	20:	
		sState := CONCAT(UDINT_TO_STRING(nState) ,' - Alaphelyzetfelvétel - Robot bekapcsolása');
		RobotOut.Control.bImmediateStop := TRUE;
		RobotOut.Control.bHold := TRUE;
		RobotOut.Control.bSafeSpeed := TRUE;
		RobotOut.Control.bEnable := TRUE;
		IF RobotIn.Status.bFault AND NOT RobotOut.Control.bReset THEN
			RobotOut.Control.bReset := TRUE;	// Ha hiba van -> Reset
		END_IF
		nState := nState + 20;

	40:
		sState := CONCAT(UDINT_TO_STRING(nState) ,' - Alaphelyzet felvétel - Robot hibatörlés');	
		IF tResetFault.Q THEN
			RobotOut.Control.bReset := FALSE;
		END_IF
		IF NOT RobotOut.Control.bReset AND NOT RobotIn.Status.bFault THEN
			nState := nState + 20;
		END_IF

	60:
		sState := CONCAT(UDINT_TO_STRING(nState) ,' - Alaphelyzet felvétel - Várakozás Robot hibatörlésre');	
		IF RobotIn.Status.bCommandEnable AND NOT RobotIn.Status.bFault THEN
			nState := nState + 20;
		END_IF
		
	80:
		sState := CONCAT(UDINT_TO_STRING(nState) ,' - Alaphelyzet felvétel - Robot Cycle Stop');
		RobotOut.Control.bCycleStop := TRUE;
		IF tStopCycle.Q THEN
			RobotOut.Control.bCycleStop := FALSE;
			nState := nState + 20;
		END_IF
	
	100:
		sState := CONCAT(UDINT_TO_STRING(nState) ,' - Alaphelyzet felvétel - Robot Cycle Start');
		RobotOut.Control.bStart := TRUE;
		IF tStartCycle.Q THEN
			RobotOut.Control.bStart := FALSE;
			nState := nState + 20;
		END_IF
		
	120: 
		sState := CONCAT(UDINT_TO_STRING(nState) ,' - Alaphelyzet felvétel - Várakozás Robot Cycle Start-ra');
		IF RobotIn.Status.bBusy AND RobotIn.Status.bProgramEnd THEN
			nState := nState + 20;
		END_IF
		
	140:
		sState := CONCAT(UDINT_TO_STRING(nState) ,' - Alaphelyzet felvétel - Alaphelyzet felvétel - Robot Busy');
		IF RobotIn.Status.bBusy THEN
			RobotOut.Control.bProdStart := TRUE;
			nState := nState + 20;
		END_IF
		
	160:
		sState := CONCAT(UDINT_TO_STRING(nState) ,' - Alaphelyzet felvétel - Robot alaphelyzetbe küldése');	
		RobotOut.Control.nProgramNumber := TO_BYTE(E_Kardex_Robot_Programs.Home);
		IF RobotOut.Control.nProgramNumber = RobotIn.Status.nProgramNumber THEN
			RobotOut.Control.nProgramNumber := 0;
			nState := nState + 20;
		END_IF
		
	180:
		sState := CONCAT(UDINT_TO_STRING(nState) ,' - Alaphelyzet felvétel - Várakozás a robotprogram végére.');	
		IF RobotIn.Status.bProgramEnd AND NOT RobotIn.Status.bProgramRun THEN
			nState := nState + 20;
		END_IF
		
	200:
		nState := 10000;
		 
(* Alaphelyzet *********************************************************************)
	10000:
		sState := CONCAT(UDINT_TO_STRING(nState) ,' - Alaphelyzet - Várakozás parancsra');
		IF eCommand = E_Kardex_Robot_Command.NoCommand THEN
			bReady := TRUE;
			bBusy := FALSE;
			bDone := FALSE;
		ELSE
			bReady := TRUE;
			bBusy := TRUE;
			bDone := FALSE;
			IF eCommand = E_Kardex_Robot_Command.Home THEN			
				nState := 11000;	
			ELSIF eCommand = E_Kardex_Robot_Command.Wait THEN	
				nState := 12000;
			ELSIF eCommand = E_Kardex_Robot_Command.Service THEN	
				nState := 13000;
			ELSIF eCommand = E_Kardex_Robot_Command.Measurement_Kardex THEN	
				nState := 14000;
			ELSIF eCommand = E_Kardex_Robot_Command.Pick_Up_Kardex THEN	
				nState := 15000;
			ELSIF eCommand = E_Kardex_Robot_Command.Put_Down_Kardex THEN	
				nState := 16000;
			ELSIF eCommand = E_Kardex_Robot_Command.Pick_Up_Mir THEN	
				nState := 17000;
			ELSIF eCommand = E_Kardex_Robot_Command.Put_Down_Mir THEN	
				nState := 18000;
			ELSIF eCommand = E_Kardex_Robot_Command.Pick_Up_Puffer THEN	
				nState := 19000;
			ELSIF eCommand = E_Kardex_Robot_Command.Put_Down_Puffer THEN	
				nState := 20000;
			ELSIF eCommand = E_Kardex_Robot_Command.Pick_Up_Strip THEN	
				nState := 21000;
			ELSIF eCommand = E_Kardex_Robot_Command.Put_Down_Strip THEN	
				nState := 22000;
			ELSIF eCommand = E_Kardex_Robot_Command.Rotate_In_Strip_3 THEN	
				nState := 23000;
			END_IF
		END_IF

{region "Move to Home"} 
	(*-----=== Move to home program végrehajtása ===-----*)
	11000:	
		sState := CONCAT(UDINT_TO_STRING(nState) ,' - Robot alaphelyzetbe küldése');	
		RobotOut.Control.nProgramNumber := TO_BYTE(E_Kardex_Robot_Programs.Home);
		IF RobotOut.Control.nProgramNumber = RobotIn.Status.nProgramNumber THEN
			RobotOut.Control.nProgramNumber := 0;
			nState := nState + 20;
		END_IF
		
	11020:
		sState := CONCAT(UDINT_TO_STRING(nState) ,' - Várakozás a robotprogram végére.');	
		IF RobotIn.Status.bProgramEnd AND NOT RobotIn.Status.bProgramRun THEN
			nState := nState + 20;
		END_IF
		
	11040:
		sState := CONCAT(UDINT_TO_STRING(nState) ,' - Várakozás mozgásparancs törlésére.');
		bReady := TRUE;
		bBusy := FALSE;
		bDone := TRUE;
		IF eCommand = E_Kardex_Robot_Command.NoCommand THEN
			nState := 10000;
		END_IF
{endregion}
	 
{region "Move to Wait"}
	(*-----=== Move to wait program végrehajtása ===-----*)
	12000:	
		sState := CONCAT(UDINT_TO_STRING(nState) ,' - Robot várakozó pozícióba küldése');	
		RobotOut.Control.nProgramNumber := TO_BYTE(E_Kardex_Robot_Programs.Park);
		IF RobotOut.Control.nProgramNumber = RobotIn.Status.nProgramNumber THEN
			RobotOut.Control.nProgramNumber := 0;
			nState := nState + 20;
		END_IF
		
	12020:
		sState := CONCAT(UDINT_TO_STRING(nState) ,' - Várakozás a robotprogram végére.');	
		IF RobotIn.Status.bProgramEnd AND NOT RobotIn.Status.bProgramRun THEN
			nState := nState + 20;
		END_IF
		
	12040:
		sState := CONCAT(UDINT_TO_STRING(nState) ,' - Várakozás mozgásparancs törlésére.');
		bReady := TRUE;
		bBusy := FALSE;
		bDone := TRUE;
		IF eCommand = E_Kardex_Robot_Command.NoCommand THEN
			nState := 10000;
		END_IF
{endregion}
	 
{region "Move to Service"}
	(*-----=== Move to service program végrehajtása ===-----*)
	13000:	
		sState := CONCAT(UDINT_TO_STRING(nState) ,' - Robot szervíz pozícióba küldése');	
		RobotOut.Control.nProgramNumber := TO_BYTE(E_Kardex_Robot_Programs.Service);
		IF RobotOut.Control.nProgramNumber = RobotIn.Status.nProgramNumber THEN
			RobotOut.Control.nProgramNumber := 0;
			nState := nState + 20;
		END_IF
		
	13020:
		sState := CONCAT(UDINT_TO_STRING(nState) ,' - Várakozás a robotprogram végére.');	
		IF RobotIn.Status.bProgramEnd AND NOT RobotIn.Status.bProgramRun THEN
			nState := nState + 20;
		END_IF
		
	13040:
		sState := CONCAT(UDINT_TO_STRING(nState) ,' - Várakozás mozgásparancs törlésére.');
		bReady := TRUE;
		bBusy := FALSE;
		bDone := TRUE;
		IF eCommand = E_Kardex_Robot_Command.NoCommand THEN
			nState := 10000;
		END_IF
{endregion}
			   
{region "Measurement Kardex"}
	(*-----=== Kardex Measurement program végrehajtása ===-----*)
	14000:	
		sState := CONCAT(UDINT_TO_STRING(nState) ,' - Kardex paletta bemérés');	
		RobotOut.Control.nProgramNumber := TO_BYTE(E_Kardex_Robot_Programs.KardexMeasurement);
		IF RobotOut.Control.nProgramNumber = RobotIn.Status.nProgramNumber THEN
			RobotOut.Control.nProgramNumber := 0;
			nState := nState + 20;
		END_IF
		
	14020:
		sState := CONCAT(UDINT_TO_STRING(nState) ,' - Várakozás a robotprogram végére.');	
		IF RobotIn.Status.bProgramEnd AND NOT RobotIn.Status.bProgramRun THEN
			nState := nState + 20;
		END_IF
		
	14040:
		sState := CONCAT(UDINT_TO_STRING(nState) ,' - Várakozás mozgásparancs törlésére.');
		bReady := TRUE;
		bBusy := FALSE;
		bDone := TRUE;
		IF eCommand = E_Kardex_Robot_Command.NoCommand THEN
			nState := 10000;
		END_IF
{endregion}
	 
{region "Pick up kardex"}
	(*-----=== Pick up Kardex program végrehajtása ===-----*)
	15000:	
		sState := CONCAT(UDINT_TO_STRING(nState) ,' - Felvétel a kardexből');
		RobotOut.Control.nKardexFloor := nKardexFloor;
		RobotOut.Control.nKardexJig := nKardexJigNumber;
		RobotOut.Control.nProgramNumber := TO_BYTE(E_Kardex_Robot_Programs.KardexPickUp);
		IF RobotOut.Control.nProgramNumber = RobotIn.Status.nProgramNumber THEN
			RobotOut.Control.nProgramNumber := 0;
			nState := nState + 20;
		END_IF
		
	15020:
		sState := CONCAT(UDINT_TO_STRING(nState) ,' - Várakozás a robotprogram végére.');	
		IF RobotIn.Status.bProgramEnd AND NOT RobotIn.Status.bProgramRun THEN
			nState := nState + 20;
		END_IF
		
	15040:
		sState := CONCAT(UDINT_TO_STRING(nState) ,' - Várakozás mozgásparancs törlésére.');
		bReady := TRUE;
		bBusy := FALSE;
		bDone := TRUE;
		IF eCommand = E_Kardex_Robot_Command.NoCommand THEN
			nState := 10000;
		END_IF
{endregion}
	 
{region "Put down kardex"}
	(*-----=== Put down Kardex program végrehajtása ===-----*)
	16000:	
		sState := CONCAT(UDINT_TO_STRING(nState) ,' - Lerakás a kardexbe');
		RobotOut.Control.nKardexFloor := nKardexFloor;
		RobotOut.Control.nKardexJig := nKardexJigNumber;
		RobotOut.Control.nProgramNumber := TO_BYTE(E_Kardex_Robot_Programs.KardexPutDown);
		IF RobotOut.Control.nProgramNumber = RobotIn.Status.nProgramNumber THEN
			RobotOut.Control.nProgramNumber := 0;
			nState := nState + 20;
		END_IF
		
	16020:
		sState := CONCAT(UDINT_TO_STRING(nState) ,' - Várakozás a robotprogram végére.');	
		IF RobotIn.Status.bProgramEnd AND NOT RobotIn.Status.bProgramRun THEN
			nState := nState + 20;
		END_IF
		
	16040:
		sState := CONCAT(UDINT_TO_STRING(nState) ,' - Várakozás mozgásparancs törlésére.');
		bReady := TRUE;
		bBusy := FALSE;
		bDone := TRUE;
		IF eCommand = E_Kardex_Robot_Command.NoCommand THEN
			nState := 10000;
		END_IF
{endregion}
	 
{region "Pick up MIR"}
	(*-----=== Pick up MIR program végrehajtása ===-----*)
	17000:	
		sState := CONCAT(UDINT_TO_STRING(nState) ,' - Felvétel a MIR-ből');
		IF nMirNumber = 1 THEN
			RobotOut.Control.nMir_1_Jig := nMir_JigNumber;							  
			RobotOut.Control.nProgramNumber := TO_BYTE(E_Kardex_Robot_Programs.Mir_1_PickUp);
		ELSIF nMirNumber = 2 THEN
			RobotOut.Control.nMir_2_Jig := nMir_JigNumber;							  
			RobotOut.Control.nProgramNumber := TO_BYTE(E_Kardex_Robot_Programs.Mir_2_PickUp);
		END_IF;
		IF RobotOut.Control.nProgramNumber = RobotIn.Status.nProgramNumber THEN
			RobotOut.Control.nProgramNumber := 0;
			nState := nState + 20;
		END_IF
		
	17020:
		sState := CONCAT(UDINT_TO_STRING(nState) ,' - Várakozás a robotprogram végére.');	
		IF RobotIn.Status.bProgramEnd AND NOT RobotIn.Status.bProgramRun THEN
			nState := nState + 20;
		END_IF
		
	17040:
		sState := CONCAT(UDINT_TO_STRING(nState) ,' - Várakozás mozgásparancs törlésére.');
		bReady := TRUE;
		bBusy := FALSE;
		bDone := TRUE;
		IF eCommand = E_Kardex_Robot_Command.NoCommand THEN
			nState := 10000;
		END_IF
{endregion}
	 
{region "Put down MIR"}
	(*-----=== Put down MIR program végrehajtása ===-----*)
	18000:	
		sState := CONCAT(UDINT_TO_STRING(nState) ,' - Lerakás a MIR-be');
		IF nMirNumber = 1 THEN
			RobotOut.Control.nMir_1_Jig := nMir_JigNumber;							  
			RobotOut.Control.nProgramNumber := TO_BYTE(E_Kardex_Robot_Programs.Mir_1_PutDown);
		ELSIF nMirNumber = 2 THEN
			RobotOut.Control.nMir_2_Jig := nMir_JigNumber;							  
			RobotOut.Control.nProgramNumber := TO_BYTE(E_Kardex_Robot_Programs.Mir_2_PutDown);
		END_IF;
		IF RobotOut.Control.nProgramNumber = RobotIn.Status.nProgramNumber THEN
			RobotOut.Control.nProgramNumber := 0;
			nState := nState + 20;
		END_IF
		
	18020:
		sState := CONCAT(UDINT_TO_STRING(nState) ,' - Várakozás a robotprogram végére.');	
		IF RobotIn.Status.bProgramEnd AND NOT RobotIn.Status.bProgramRun THEN
			nState := nState + 20;
		END_IF
		
	18040:
		sState := CONCAT(UDINT_TO_STRING(nState) ,' - Várakozás mozgásparancs törlésére.');
		bReady := TRUE;
		bBusy := FALSE;
		bDone := TRUE;
		IF eCommand = E_Kardex_Robot_Command.NoCommand THEN
			nState := 10000;
		END_IF
{endregion}
								   
{region "Pick up Puffer"}
	(*-----=== Pick up Puffer program végrehajtása ===-----*)
	19000:	
		sState := CONCAT(UDINT_TO_STRING(nState) ,' - Felvétel a pufferből');
		RobotOut.Control.nPuffer := nPufferNumber;
		RobotOut.Control.nProgramNumber := TO_BYTE(E_Kardex_Robot_Programs.PufferPickUp);
		IF RobotOut.Control.nProgramNumber = RobotIn.Status.nProgramNumber THEN
			RobotOut.Control.nProgramNumber := 0;
			nState := nState + 20;
		END_IF
		
	19020:
		sState := CONCAT(UDINT_TO_STRING(nState) ,' - Várakozás a robotprogram végére.');	
		IF RobotIn.Status.bProgramEnd AND NOT RobotIn.Status.bProgramRun THEN
			nState := nState + 20;
		END_IF
		
	19040:
		sState := CONCAT(UDINT_TO_STRING(nState) ,' - Várakozás mozgásparancs törlésére.');
		bReady := TRUE;
		bBusy := FALSE;
		bDone := TRUE;
		IF eCommand = E_Kardex_Robot_Command.NoCommand THEN
			nState := 10000;
		END_IF
{endregion}
	 
{region "Put down Puffer"}
	(*-----=== Put down Puffer program végrehajtása ===-----*)
	20000:	
		sState := CONCAT(UDINT_TO_STRING(nState) ,' - Lerakás a pufferbe');
		RobotOut.Control.nPuffer := nPufferNumber;
		RobotOut.Control.nProgramNumber := TO_BYTE(E_Kardex_Robot_Programs.PufferPutDown);
		IF RobotOut.Control.nProgramNumber = RobotIn.Status.nProgramNumber THEN
			RobotOut.Control.nProgramNumber := 0;
			nState := nState + 20;
		END_IF
		
	20020:
		sState := CONCAT(UDINT_TO_STRING(nState) ,' - Várakozás a robotprogram végére.');	
		IF RobotIn.Status.bProgramEnd AND NOT RobotIn.Status.bProgramRun THEN
			nState := nState + 20;
		END_IF
		
	20040:
		sState := CONCAT(UDINT_TO_STRING(nState) ,' - Várakozás mozgásparancs törlésére.');
		bReady := TRUE;
		bBusy := FALSE;
		bDone := TRUE;
		IF eCommand = E_Kardex_Robot_Command.NoCommand THEN
			nState := 10000;
		END_IF
{endregion}
											 
{region "Pick up Strip"}
	(*-----=== Pick up Strip program végrehajtása ===-----*)
	21000:	
		sState := CONCAT(UDINT_TO_STRING(nState) ,' - Felvétel a szalagról');
		IF nStripNumber = 1 THEN					  
			RobotOut.Control.nProgramNumber := TO_BYTE(E_Kardex_Robot_Programs.Strip_1_PickUp);
		ELSIF nStripNumber = 2 THEN						  
			RobotOut.Control.nProgramNumber := TO_BYTE(E_Kardex_Robot_Programs.Strip_2_PickUp);
		ELSIF nStripNumber = 3 THEN						  
			RobotOut.Control.nProgramNumber := TO_BYTE(E_Kardex_Robot_Programs.Strip_3_PickUp);
		END_IF;
		IF RobotOut.Control.nProgramNumber = RobotIn.Status.nProgramNumber THEN
			RobotOut.Control.nProgramNumber := 0;
			nState := nState + 20;
		END_IF
		
	21020:
		sState := CONCAT(UDINT_TO_STRING(nState) ,' - Várakozás a robotprogram végére.');	
		IF RobotIn.Status.bProgramEnd AND NOT RobotIn.Status.bProgramRun THEN
			nState := nState + 20;
		END_IF
		
	21040:
		sState := CONCAT(UDINT_TO_STRING(nState) ,' - Várakozás mozgásparancs törlésére.');
		bReady := TRUE;
		bBusy := FALSE;
		bDone := TRUE;
		IF eCommand = E_Kardex_Robot_Command.NoCommand THEN
			nState := 10000;
		END_IF
{endregion}
	 
{region "Put down Strip"}
	(*-----=== Put down Strip program végrehajtása ===-----*)
	22000:	
		sState := CONCAT(UDINT_TO_STRING(nState) ,' - Lerakás a szalagra');
		IF nStripNumber = 1 THEN					  
			RobotOut.Control.nProgramNumber := TO_BYTE(E_Kardex_Robot_Programs.Strip_1_PutDown);
		ELSIF nStripNumber = 2 THEN						  
			RobotOut.Control.nProgramNumber := TO_BYTE(E_Kardex_Robot_Programs.Strip_2_PutDown);
		ELSIF nStripNumber = 3 THEN						  
			RobotOut.Control.nProgramNumber := TO_BYTE(E_Kardex_Robot_Programs.Strip_3_PutDown);
		END_IF;
		IF RobotOut.Control.nProgramNumber = RobotIn.Status.nProgramNumber THEN
			RobotOut.Control.nProgramNumber := 0;
			nState := nState + 20;
		END_IF
		
	22020:
		sState := CONCAT(UDINT_TO_STRING(nState) ,' - Várakozás a robotprogram végére.');	
		IF RobotIn.Status.bProgramEnd AND NOT RobotIn.Status.bProgramRun THEN
			nState := nState + 20;
		END_IF
		
	22040:
		sState := CONCAT(UDINT_TO_STRING(nState) ,' - Várakozás mozgásparancs törlésére.');
		bReady := TRUE;
		bBusy := FALSE;
		bDone := TRUE;
		IF eCommand = E_Kardex_Robot_Command.NoCommand THEN
			nState := 10000;
		END_IF
{endregion}
{region "Rotate in strip 3"}
	(*-----=== Rotate in strip 3 program végrehajtása ===-----*)
	23000:	
		sState := CONCAT(UDINT_TO_STRING(nState) ,' - Forgatás a 3-as szalagon');	
		RobotOut.Control.nProgramNumber := TO_BYTE(E_Kardex_Robot_Programs.Strip_3_Rotate);
		IF RobotOut.Control.nProgramNumber = RobotIn.Status.nProgramNumber THEN
			RobotOut.Control.nProgramNumber := 0;
			nState := nState + 20;
		END_IF
		
	23020:
		sState := CONCAT(UDINT_TO_STRING(nState) ,' - Várakozás a robotprogram végére.');	
		IF RobotIn.Status.bProgramEnd AND NOT RobotIn.Status.bProgramRun THEN
			nState := nState + 20;
		END_IF
		
	23040:
		sState := CONCAT(UDINT_TO_STRING(nState) ,' - Várakozás mozgásparancs törlésére.');
		bReady := TRUE;
		bBusy := FALSE;
		bDone := TRUE;
		IF eCommand = E_Kardex_Robot_Command.NoCommand THEN
			nState := 10000;
		END_IF
{endregion}
	 
{region "Pendant mode"}
(* Pendant mód *********************************************************************)
	150000:	sState := CONCAT(UDINT_TO_STRING(nState) ,' - Pendant mód');
			IF NOT bPendantMode THEN
				RobotOut.Control.bImmediateStop := FALSE;
				RobotOut.Control.bHold := FALSE;
				RobotOut.Control.bZoneEnable := FALSE;
				RobotOut.Control.bEnable := FALSE;
				nState := 0;
			ELSE
				RobotOut.Control.bEnable := TRUE;
				RobotOut.Control.bHold := TRUE;
				RobotOut.Control.bZoneEnable := TRUE;
				RobotOut.Control.bImmediateStop := TRUE;
			END_IF
{endregion}
		
(* Hibakezelés *********************************************************************)
	200000:	sState := CONCAT(UDINT_TO_STRING(nState) ,CONCAT(' - Hiba, ebből az állapotból: ' ,sState));
			bReady := FALSE;
			bBusy := FALSE;	
			nState := nState + 20;

(* Hibakezelés *********************************************************************)
	200020:	
			IF bAck THEN			
				nState := nState + 20;
			END_IF
			
	200040: 
			RobotOut.Control.bImmediateStop := TRUE;
			RobotOut.Control.bReset := TRUE;
			RobotOut.Control.bNotCorrectPrg_Reset := TRUE;
			RobotOut.Control.bNotProductOnRobot_Reset := TRUE;
			RobotOut.Control.bProductOnRobot_Reset := TRUE;
			RobotOut.Control.bGripperOpenError_Reset := TRUE;
			RobotOut.Control.bGripperCloseError_Reset := TRUE;
			RobotOut.Control.bPartPresentError_Reset := TRUE;
			RobotOut.Control.bNotCorrectKardexFloor_Reset := TRUE;
			RobotOut.Control.bNotCorrectKardexJig_Reset := TRUE;
			RobotOut.Control.bNotCorrectMir_Reset := TRUE;
			RobotOut.Control.bNotCorrectPuffer_Reset := TRUE;
			nState := nState + 20;
			
	200060:
			IF 	NOT RobotIn.Status.bNoPneumatics AND
				NOT RobotIn.Status.bNotCorrectPrg AND
				NOT RobotIn.Status.bNotProductOnRobot AND
				NOT RobotIn.Status.bProductOnRobot AND
				NOT RobotIn.Status.bGripperOpenError AND
				NOT RobotIn.Status.bGripperCloseError AND
				NOT RobotIn.Status.bPartPresentError AND
				NOT	RobotIn.Status.bNotCorrectKardexFloor AND
				NOT RobotIn.Status.bNotCorrectKardexJig AND
				NOT RobotIn.Status.bNotCorrectMir AND
				NOT RobotIn.Status.bNotCorrectPuffer														 
			THEN
				nState := nState + 20;
			END_IF	
			
	200080:
			RobotOut.Control.bReset := FALSE;
			RobotOut.Control.bNotCorrectPrg_Reset := FALSE;
			RobotOut.Control.bNotProductOnRobot_Reset := FALSE;
			RobotOut.Control.bProductOnRobot_Reset := FALSE;
			RobotOut.Control.bGripperOpenError_Reset := FALSE;
			RobotOut.Control.bGripperCloseError_Reset := FALSE;
			RobotOut.Control.bPartPresentError_Reset := FALSE;
			RobotOut.Control.bNotCorrectKardexFloor_Reset := FALSE;
			RobotOut.Control.bNotCorrectKardexJig_Reset := FALSE;
			RobotOut.Control.bNotCorrectMir_Reset := FALSE;
			RobotOut.Control.bNotCorrectPuffer_Reset := FALSE;
			bErrNotReady := FALSE;
			bErrBaseTimeout := FALSE;
			nState := 0;
ELSE
	sState := CONCAT(UDINT_TO_STRING(nState) ,' - Nem használt állapot');
END_CASE	


(*Hiba string*)
IF bError THEN
	sError := sName;
	FOR i:=0 TO nMaxAlarmNr DO
		IF arrAlarms[i] THEN
			IF (fbAlarmArray[i].eConfirmationState <> 2 AND fbAlarmArray[i].nTimeCleared <> 0 AND fbAlarmArray[i].nTimeConfirmed <> 0) OR //Ha már volt alarm, akkor van bennük érték
				(fbAlarmArray[i].eConfirmationState = 1 AND fbAlarmArray[i].nTimeCleared = 0 AND fbAlarmArray[i].nTimeConfirmed = 0)	//Első futás esetén
			THEN
				fbAlarmArray[i].Raise(0);
			END_IF
		END_IF
	END_FOR 
ELSE
	sError := '';
END_IF

(*Hiba kezelés Tc3_EventLogger*)
IF NOT bIsInitalized THEN
	bIsInitalized := TRUE;
	FOR i:=0 TO nMaxAlarmNr DO
		fbAlarmArray[i].CreateEx(stEventArray[i], TRUE, 0);
	END_FOR
END_IF

(*Hiba törlés (nyugtázott és megszűnt)*)
FOR i:=0 TO nMaxAlarmNr DO
	IF fbAlarmArray[i].eConfirmationState = 3 AND NOT bError THEN
		fbAlarmArray[i].Clear(0, FALSE);
	END_IF
END_FOR

END_FUNCTION_BLOCK

// ---- POUs/ConveyorSystem.TcPOU
PROGRAM ConveyorSystem
VAR
	(*ID_200*)
	rtStartReaders	: R_TRIG;
	bStartReaders	: BOOL;	
	i				: INT := 1;
	ch				: BYTE := 1;
	j				: INT := 1;
	k				: INT := 1;
	FixCode			: ARRAY [0..4] OF BYTE;
	TestData 		: ARRAY [0..7] OF BYTE;
	(*Head Data*)

	bTestQuit			: BOOL;
	bTestERFC			: BOOL;
	bTestERWS			: BOOL;
	bTestCT				: BOOL;
	bTestReset			: BOOL;
	bTestChannel		: BYTE := 1;
	
	bTestSWFC			: BOOL;
	bTestSWWS			: BOOL;
	
	pvPaletteData		: PVOID;
	nRouterIndex		: BYTE;
END_VAR
VAR CONSTANT
	arrRFIDs			: ARRAY[1..17] OF ST_Active_RFIDs := [	(RFID := 1, CH := 2),	//RF 1
																(RFID := 1, CH := 1),	//RF 2
																(RFID := 2, CH := 1),	//RF 3
																(RFID := 2, CH := 2),	//RF 4
																(RFID := 3, CH := 1),	//RF 5
																(RFID := 3, CH := 2),	//RF 6
																(RFID := 4, CH := 1),	//RF 7
																(RFID := 4, CH := 2),	//RF 8
																(RFID := 5, CH := 2),	//RF 9
																(RFID := 5, CH := 1),	//RF 10
																(RFID := 6, CH := 1),	//RF 11
																(RFID := 7, CH := 1),	//RF 13
																(RFID := 9, CH := 2),	//RF 15
																(RFID := 8, CH := 2),	//RF 16
																(RFID := 8, CH := 1),	//RF 17
																(RFID := 10, CH := 1),	//RF 18
																(RFID := 9, CH := 1)];	//RF 19
END_VAR

Cylinders();
Stoppers();
Motors();
Lift();
ID_200();
ID_200_Test();
Routers();

ACTION Cylinders:
fbZ1(
	sName:= 'Kiemelő 1A', 
	bEn:= i_bLO1_Main, 
	bEHA:= NOT bManualMode, 
	nEHMode:= 2, 
	bDisableManualCmd:= NOT bManualMode, 
	bAck:= bAckP, 
	i_bBasePos:= i_stSensorHub_7.Channel_1 AND i_stSensorHub_7.Channel_3, 
	i_bWorkPos:= i_stSensorHub_7.Channel_0 AND i_stSensorHub_7.Channel_2, 
	sSourceName:= , 
	stBasePosEvent:= , 
	stWorkPosEvent:= , 
	q_bBasePos=> GVL_ConveyorSystem.q_bZ1_12, 
	q_bWorkPos=> GVL_ConveyorSystem.q_bZ1_14);
	
fbZ2(
	sName:= 'Kiemelő 1B', 
	bEn:= i_bLO1_Main, 
	bEHA:= NOT bManualMode, 
	nEHMode:= 2, 
	bDisableManualCmd:= NOT bManualMode, 
	bAck:= bAckP, 
	i_bBasePos:= i_stSensorHub_6.Channel_1 AND i_stSensorHub_6.Channel_3, 
	i_bWorkPos:= i_stSensorHub_6.Channel_0 AND i_stSensorHub_6.Channel_2, 
	sSourceName:= , 
	stBasePosEvent:= , 
	stWorkPosEvent:= , 
	q_bBasePos=> GVL_ConveyorSystem.q_bZ2_12, 
	q_bWorkPos=> GVL_ConveyorSystem.q_bZ2_14);
	
fbZ3(
	sName:= 'Kiemelő 2A', 
	bEn:= i_bLO1_Main, 
	bEHA:= NOT bManualMode, 
	nEHMode:= 2, 
	bDisableManualCmd:= NOT bManualMode, 
	bAck:= bAckP, 
	i_bBasePos:= i_stSensorHub_10.Channel_0 AND i_stSensorHub_10.Channel_2, 
	i_bWorkPos:= i_stSensorHub_10.Channel_1 AND i_stSensorHub_10.Channel_3, 
	sSourceName:= , 
	stBasePosEvent:= , 
	stWorkPosEvent:= , 
	q_bBasePos=> GVL_ConveyorSystem.q_bZ3_12, 
	q_bWorkPos=> GVL_ConveyorSystem.q_bZ3_14);
	
fbZ4(
	sName:= 'Kiemelő 2B', 
	bEn:= i_bLO1_Main, 
	bEHA:= NOT bManualMode, 
	nEHMode:= 2, 
	bDisableManualCmd:= NOT bManualMode, 
	bAck:= bAckP, 
	i_bBasePos:= i_stSensorHub_11.Channel_0 AND i_stSensorHub_11.Channel_2, 
	i_bWorkPos:= i_stSensorHub_11.Channel_1 AND i_stSensorHub_11.Channel_3, 
	sSourceName:= , 
	stBasePosEvent:= , 
	stWorkPosEvent:= , 
	q_bBasePos=> GVL_ConveyorSystem.q_bZ4_12, 
	q_bWorkPos=> GVL_ConveyorSystem.q_bZ4_14);
	
fbZ5(
	sName:= 'Kiemelő 3A', 
	bEn:= i_bLO1_Main, 
	bEHA:= NOT bManualMode, 
	nEHMode:= 2, 
	bDisableManualCmd:= NOT bManualMode, 
	bAck:= bAckP, 
	i_bBasePos:= i_stSensorHub_14.Channel_1 AND i_stSensorHub_14.Channel_3, 
	i_bWorkPos:= i_stSensorHub_14.Channel_0 AND i_stSensorHub_14.Channel_2, 
	sSourceName:= , 
	stBasePosEvent:= , 
	stWorkPosEvent:= , 
	q_bBasePos=> GVL_ConveyorSystem.q_bZ5_12, 
	q_bWorkPos=> GVL_ConveyorSystem.q_bZ5_14);
	
fbZ6(
	sName:= 'Kiemelő 3B', 
	bEn:= i_bLO1_Main, 
	bEHA:= NOT bManualMode, 
	nEHMode:= 2, 
	bDisableManualCmd:= NOT bManualMode, 
	bAck:= bAckP, 
	i_bBasePos:= i_stSensorHub_15.Channel_1 AND i_stSensorHub_15.Channel_3, 
	i_bWorkPos:= i_stSensorHub_15.Channel_0 AND i_stSensorHub_15.Channel_2, 
	sSourceName:= , 
	stBasePosEvent:= , 
	stWorkPosEvent:= , 
	q_bBasePos=> GVL_ConveyorSystem.q_bZ6_12, 
	q_bWorkPos=> GVL_ConveyorSystem.q_bZ6_14);
	
fbZ7(
	sName:= 'Paletta megfogó 1A', 
	bEn:= i_bLO1_Main, 
	bEHA:= NOT bManualMode, 
	nEHMode:= 2, 
	bDisableManualCmd:= NOT bManualMode, 
	bAck:= bAckP, 
	i_bBasePos:= i_stSensorHub_7.Channel_4, 
	i_bWorkPos:= i_stSensorHub_7.Channel_5, 
	sSourceName:= , 
	stBasePosEvent:= , 
	stWorkPosEvent:= , 
	q_bBasePos=> GVL_ConveyorSystem.q_bZ7_12, 
	q_bWorkPos=> GVL_ConveyorSystem.q_bZ7_14);
	
fbZ8(
	sName:= 'Paletta megfogó 1B', 
	bEn:= i_bLO1_Main, 
	bEHA:= NOT bManualMode, 
	nEHMode:= 2, 
	bDisableManualCmd:= NOT bManualMode, 
	bAck:= bAckP, 
	i_bBasePos:= i_stSensorHub_6.Channel_4, 
	i_bWorkPos:= i_stSensorHub_6.Channel_5, 
	sSourceName:= , 
	stBasePosEvent:= , 
	stWorkPosEvent:= , 
	q_bBasePos=> GVL_ConveyorSystem.q_bZ8_12, 
	q_bWorkPos=> GVL_ConveyorSystem.q_bZ8_14);
	
fbZ9(
	sName:= 'Paletta megfogó 2A', 
	bEn:= i_bLO1_Main, 
	bEHA:= NOT bManualMode, 
	nEHMode:= 2, 
	bDisableManualCmd:= NOT bManualMode, 
	bAck:= bAckP, 
	i_bBasePos:= i_stSensorHub_10.Channel_4, 
	i_bWorkPos:= i_stSensorHub_10.Channel_5, 
	sSourceName:= , 
	stBasePosEvent:= , 
	stWorkPosEvent:= , 
	q_bBasePos=> GVL_ConveyorSystem.q_bZ9_12, 
	q_bWorkPos=> GVL_ConveyorSystem.q_bZ9_14);
	
fbZ10(
	sName:= 'Paletta megfogó 2B', 
	bEn:= i_bLO1_Main, 
	bEHA:= NOT bManualMode, 
	nEHMode:= 2, 
	bDisableManualCmd:= NOT bManualMode, 
	bAck:= bAckP, 
	i_bBasePos:= i_stSensorHub_11.Channel_4, 
	i_bWorkPos:= i_stSensorHub_11.Channel_5, 
	sSourceName:= , 
	stBasePosEvent:= , 
	stWorkPosEvent:= , 
	q_bBasePos=> GVL_ConveyorSystem.q_bZ10_12, 
	q_bWorkPos=> GVL_ConveyorSystem.q_bZ10_14);
	
fbZ11(
	sName:= 'Paletta megfogó 3A', 
	bEn:= i_bLO1_Main, 
	bEHA:= NOT bManualMode, 
	nEHMode:= 2, 
	bDisableManualCmd:= NOT bManualMode, 
	bAck:= bAckP, 
	i_bBasePos:= i_stSensorHub_14.Channel_4, 
	i_bWorkPos:= i_stSensorHub_14.Channel_5, 
	sSourceName:= , 
	stBasePosEvent:= , 
	stWorkPosEvent:= , 
	q_bBasePos=> GVL_ConveyorSystem.q_bZ11_12, 
	q_bWorkPos=> GVL_ConveyorSystem.q_bZ11_14);
	
fbZ12(
	sName:= 'Paletta megfogó 3B', 
	bEn:= i_bLO1_Main, 
	bEHA:= NOT bManualMode, 
	nEHMode:= 2, 
	bDisableManualCmd:= NOT bManualMode, 
	bAck:= bAckP, 
	i_bBasePos:= i_stSensorHub_15.Channel_4, 
	i_bWorkPos:= i_stSensorHub_15.Channel_5, 
	sSourceName:= , 
	stBasePosEvent:= , 
	stWorkPosEvent:= , 
	q_bBasePos=> GVL_ConveyorSystem.q_bZ12_12, 
	q_bWorkPos=> GVL_ConveyorSystem.q_bZ12_14);
	
fbZ13(
	sName:= 'Útválasztó kihordó visszafordító', 
	bEn:= i_bLO1_Main, 
	bEHA:= NOT bManualMode, 
	nEHMode:= , 
	bDisableManualCmd:= NOT bManualMode, 
	bAck:= bAckP, 
	i_bBasePos:= i_stSensorHub_16.Channel_4, 
	i_bWorkPos:= i_stSensorHub_16.Channel_3, 
	sSourceName:= , 
	stBasePosEvent:= , 
	stWorkPosEvent:= , 
	q_bBasePos=> GVL_ConveyorSystem.q_bZ13_12, 
	q_bWorkPos=> GVL_ConveyorSystem.q_bZ13_14);
	
fbZ14(
	sName:= 'Útválasztó CNC2 puffer behordás', 
	bEn:= i_bLO1_Main, 
	bEHA:= NOT bManualMode, 
	nEHMode:= 2, 
	bDisableManualCmd:= NOT bManualMode, 
	bAck:= bAckP, 
	i_bBasePos:= i_stSensorHub_12.Channel_0, 
	i_bWorkPos:= i_stSensorHub_12.Channel_1, 
	sSourceName:= , 
	stBasePosEvent:= , 
	stWorkPosEvent:= , 
	q_bBasePos=> GVL_ConveyorSystem.q_bZ14_12, 
	q_bWorkPos=> GVL_ConveyorSystem.q_bZ14_14);
	
fbZ15(
	sName:= 'Útválasztó CNC3 puffer kihordás', 
	bEn:= i_bLO1_Main, 
	bEHA:= NOT bManualMode, 
	nEHMode:= 2, 
	bDisableManualCmd:= NOT bManualMode, 
	bAck:= bAckP, 
	i_bBasePos:= i_stSensorHub_13.Channel_0, 
	i_bWorkPos:= i_stSensorHub_13.Channel_1, 
	sSourceName:= , 
	stBasePosEvent:= , 
	stWorkPosEvent:= , 
	q_bBasePos=> GVL_ConveyorSystem.q_bZ15_12, 
	q_bWorkPos=> GVL_ConveyorSystem.q_bZ15_14);
	
fbZ16(
	sName:= 'Útválasztó CNC2 puffer behordás', 
	bEn:= i_bLO1_Main, 
	bEHA:= NOT bManualMode, 
	nEHMode:= 2, 
	bDisableManualCmd:= NOT bManualMode, 
	bAck:= bAckP, 
	i_bBasePos:= i_stSensorHub_8.Channel_1, 
	i_bWorkPos:= i_stSensorHub_8.Channel_0, 
	sSourceName:= , 
	stBasePosEvent:= , 
	stWorkPosEvent:= , 
	q_bBasePos=> GVL_ConveyorSystem.q_bZ16_12, 
	q_bWorkPos=> GVL_ConveyorSystem.q_bZ16_14);
	
fbZ17(
	sName:= 'Útválasztó CNC2 puffer kihordás', 
	bEn:= i_bLO1_Main, 
	bEHA:= NOT bManualMode, 
	nEHMode:= 2, 
	bDisableManualCmd:= NOT bManualMode, 
	bAck:= bAckP, 
	i_bBasePos:= i_stSensorHub_8.Channel_3, 
	i_bWorkPos:= i_stSensorHub_8.Channel_2, 
	sSourceName:= , 
	stBasePosEvent:= , 
	stWorkPosEvent:= , 
	q_bBasePos=> GVL_ConveyorSystem.q_bZ17_12, 
	q_bWorkPos=> GVL_ConveyorSystem.q_bZ17_14);
	
fbZ18(
	sName:= 'Útválasztó CNC1 puffer behordás', 
	bEn:= i_bLO1_Main, 
	bEHA:= NOT bManualMode, 
	nEHMode:= 2, 
	bDisableManualCmd:= NOT bManualMode, 
	bAck:= bAckP, 
	i_bBasePos:= i_stSensorHub_5.Channel_1, 
	i_bWorkPos:= i_stSensorHub_5.Channel_0, 
	sSourceName:= , 
	stBasePosEvent:= , 
	stWorkPosEvent:= , 
	q_bBasePos=> GVL_ConveyorSystem.q_bZ18_12, 
	q_bWorkPos=> GVL_ConveyorSystem.q_bZ18_14);
	
fbZ19(
	sName:= 'Útválasztó CNC1 puffer kihordás', 
	bEn:= i_bLO1_Main, 
	bEHA:= NOT bManualMode, 
	nEHMode:= 2, 
	bDisableManualCmd:= NOT bManualMode, 
	bAck:= bAckP, 
	i_bBasePos:= i_stSensorHub_5.Channel_2, 
	i_bWorkPos:= i_stSensorHub_5.Channel_3, 
	sSourceName:= , 
	stBasePosEvent:= , 
	stWorkPosEvent:= , 
	q_bBasePos=> GVL_ConveyorSystem.q_bZ19_12, 
	q_bWorkPos=> GVL_ConveyorSystem.q_bZ19_14);
	
fbZ20(
	sName:= 'Útválasztó CNC1 előtt', 
	bEn:= i_bLO1_Main, 
	bEHA:= NOT bManualMode, 
	nEHMode:= 2, 
	bDisableManualCmd:= NOT bManualMode, 
	bAck:= bAckP, 
	i_bBasePos:= i_stSensorHub_1.Channel_0, 
	i_bWorkPos:= i_stSensorHub_1.Channel_1, 
	sSourceName:= , 
	stBasePosEvent:= , 
	stWorkPosEvent:= , 
	q_bBasePos=> GVL_ConveyorSystem.q_bZ20_12, 
	q_bWorkPos=> GVL_ConveyorSystem.q_bZ20_14);
	
fbZ21(
	sName:= 'Útválasztó kihordás', 
	bEn:= i_bLO1_Main, 
	bEHA:= NOT bManualMode, 
	nEHMode:= , 
	bDisableManualCmd:= NOT bManualMode, 
	bAck:= bAckP, 
	i_bBasePos:= i_stSensorHub_1.Channel_4, 
	i_bWorkPos:= i_stSensorHub_1.Channel_5, 
	sSourceName:= , 
	stBasePosEvent:= , 
	stWorkPosEvent:= , 
	q_bBasePos=> GVL_ConveyorSystem.q_bZ21_12, 
	q_bWorkPos=> GVL_ConveyorSystem.q_bZ21_14);
END_ACTION

ACTION ID_200:
rtStartReaders(CLK:= NOT bManualModeVise OR i_bLO1_Main, Q=> );
IF rtStartReaders.Q THEN
	i := 1;
	bStartReaders := TRUE;
END_IF

IF bStartReaders THEN
	IF fbRFID_Readers[arrRFIDs[i].RFID].EncReadFixCode(arrRFIDs[i].CH) THEN
		i := i + 1;
	END_IF
	IF i > 17 THEN
		bStartReaders := FALSE;
	END_IF
END_IF

FOR j:=1 TO 10 DO
	fbRFID_Readers[j]();
END_FOR
END_ACTION

ACTION ID_200_Test:
(*-----=== Test ===-----*)
IF bTestReset THEN
	IF fbRFID_Readers[k].Reset() THEN
		bTestReset := FALSE;
	END_IF
END_IF

IF bTestQuit THEN
	IF fbRFID_Readers[k].Quit(bTestChannel) THEN
		bTestQuit := FALSE;
	END_IF
END_IF

IF bTestERWS THEN
	IF fbRFID_Readers[k].EncReadWords(bTestChannel, 5, ) THEN
		bTestERWS := FALSE;
	END_IF
END_IF

IF bTestERFC THEN
	IF fbRFID_Readers[k].EncReadFixCode(bTestChannel) THEN
		bTestERFC := FALSE;
	END_IF
END_IF

IF bTestCT THEN
	IF fbRFID_Readers[k].ChangeTag(			Channel := bTestChannel,
									CarrierType := E_CarrierType.MDT_28) THEN
		bTestCT := FALSE;
	END_IF
END_IF

//v1
IF bTestSWFC THEN
	IF fbRFID_Readers[k].SinWriteFixCode(	Channel := bTestChannel,
													Data := FixCode) THEN
		bTestSWFC := FALSE;
	END_IF
END_IF

//v2
//IF bTestSWFC THEN
//	IF fbId200_1.SinWriteFixCode(	Channel := bTestChannel,
//									Fixlen := uFixLength,
//									CarrierType := E_CarrierType.MDT_28,
//									Data := TestData,
//									DataLength := 5) THEN
//		bTestSWFC := FALSE;
//	END_IF
//END_IF

IF bTestSWWS THEN
	IF fbRFID_Readers[k].SinWriteWords(		Channel := bTestChannel,
									1,
									Data := TestData,
									DataLength := 5) THEN
		bTestSWWS := FALSE;
	END_IF
END_IF
END_ACTION

ACTION Lift:
fbLift_1A(
	bEnable:= i_bLO1_Main, 
	bErrorAck:= bAckP, 
	bManualMode:= bManualMode,
	bStepEnable:= bStepEnable, 
	bBeforeStopperSent:= fbS19.bPalletSent,
	stTagData:= fbRFID_Readers[1].Ch2_TagData,
	nReqTarget:= 2, 							// CNC1-re váró palettákat fogad
	fbLift:= ADR(fbZ1), 
	fbLock:= ADR(fbZ7), 
	fbStopper:= ADR(fbS1),
	arrPaletteData:= ADR(arrPalette));

fbLift_1B(
	bEnable:= i_bLO1_Main, 
	bErrorAck:= bAckP, 
	bManualMode:= bManualMode,
	bStepEnable:= bStepEnable, 
	bBeforeStopperSent:= fbS1.bPalletSent,
	stTagData:= fbRFID_Readers[1].Ch1_TagData, 
	nReqTarget:= 2,  							// CNC1-re váró palettákat fogad
	fbLift:= ADR(fbZ2), 
	fbLock:= ADR(fbZ8), 
	fbStopper:= ADR(fbS2),
	arrPaletteData:= ADR(arrPalette));

fbLift_2A(
	bEnable:= i_bLO1_Main, 
	bErrorAck:= bAckP, 
	bManualMode:= bManualMode,
	bStepEnable:= bStepEnable, 
	bBeforeStopperSent:= fbS17.bPalletSent,
	stTagData:= fbRFID_Readers[2].Ch1_TagData, 
	nReqTarget:= 4,  							// CNC2-re váró palettákat fogad
	fbLift:= ADR(fbZ3), 
	fbLock:= ADR(fbZ9), 
	fbStopper:= ADR(fbS3),
	arrPaletteData:= ADR(arrPalette));

fbLift_2B(
	bEnable:= i_bLO1_Main, 
	bErrorAck:= bAckP, 
	bManualMode:= bManualMode,
	bStepEnable:= bStepEnable, 
	bBeforeStopperSent:= fbS3.bPalletSent,
	stTagData:= fbRFID_Readers[2].Ch2_TagData, 
	nReqTarget:= 4,  							// CNC2-re váró palettákat fogad
	fbLift:= ADR(fbZ4), 
	fbLock:= ADR(fbZ10), 
	fbStopper:= ADR(fbS4),
	arrPaletteData:= ADR(arrPalette));

fbLift_3A(
	bEnable:= i_bLO1_Main, 
	bErrorAck:= bAckP, 
	bManualMode:= bManualMode,
	bStepEnable:= bStepEnable, 
	bBeforeStopperSent:= fbS13.bPalletSent,
	stTagData:= fbRFID_Readers[3].Ch1_TagData, 
	nReqTarget:= 6,  							// CNC3-ra váró palettákat fogad
	fbLift:= ADR(fbZ5), 
	fbLock:= ADR(fbZ11), 
	fbStopper:= ADR(fbS5),
	arrPaletteData:= ADR(arrPalette));

fbLift_3B(
	bEnable:= i_bLO1_Main, 
	bErrorAck:= bAckP, 
	bManualMode:= bManualMode,
	bStepEnable:= bStepEnable, 
	bBeforeStopperSent:= fbS5.bPalletSent,
	stTagData:= fbRFID_Readers[3].Ch2_TagData, 
	nReqTarget:= 6,  							// CNC3-ra váró palettákat fogad
	fbLift:= ADR(fbZ6), 
	fbLock:= ADR(fbZ12), 
	fbStopper:= ADR(fbS6),
	arrPaletteData:= ADR(arrPalette));
END_ACTION

ACTION Motors:
IF NOT bManualMode THEN
	fbConveyor_1.bConveyorOnL := i_bLO1_Main;
	fbConveyor_2.bConveyorOnL := i_bLO1_Main;
	fbConveyor_3.bConveyorOnL := i_bLO1_Main;
	fbConveyor_4.bConveyorOnL := i_bLO1_Main;
	fbConveyor_5.bConveyorOnL := i_bLO1_Main;
	fbConveyor_6.bConveyorOnL := i_bLO1_Main;
	fbConveyor_7.bConveyorOnL := i_bLO1_Main;
	fbConveyor_8.bConveyorOnL := i_bLO1_Main;
	fbConveyor_9.bConveyorOnL := i_bLO1_Main;
	fbConveyor_10.bConveyorOnL := i_bLO1_Main;
	fbConveyor_11.bConveyorOnL := i_bLO1_Main;
END_IF

fbConveyor_1(
	sName:= 'Konveyor motor M1', 
	bEn:= i_bLO1_Main, 
	bEHA:= NOT bManualMode, 
	bDisableManualCmd:= NOT bManualMode, 
	bConveyorOnL:= , 
	bConveyorOnR:= , 
	timReset:= , 
	bAck:= bAckP, 
	i_bConveyorOK:= i_bConveyor_1_Ok, 
	stStartEvent:= , 
	stRunEvent:= , 
	bMotorOn=> , 
	bError=> , 
	sError=> , 
	q_bConveyorOnL=> q_bConveyor_1, 
	q_bConveyorOnR=> , 
	q_bConveyorRst=> );

fbConveyor_2(
	sName:= 'Konveyor motor M2', 
	bEn:= i_bLO1_Main, 
	bEHA:= NOT bManualMode, 
	bDisableManualCmd:= NOT bManualMode, 
	bConveyorOnL:= , 
	bConveyorOnR:= , 
	timReset:= , 
	bAck:= bAckP, 
	i_bConveyorOK:= i_bConveyor_2_Ok, 
	stStartEvent:= , 
	stRunEvent:= , 
	bMotorOn=> , 
	bError=> , 
	sError=> , 
	q_bConveyorOnL=> q_bConveyor_2, 
	q_bConveyorOnR=> , 
	q_bConveyorRst=> );

fbConveyor_3(
	sName:= 'Konveyor motor M3', 
	bEn:= i_bLO1_Main, 
	bEHA:= NOT bManualMode, 
	bDisableManualCmd:= NOT bManualMode, 
	bConveyorOnL:= , 
	bConveyorOnR:= , 
	timReset:= , 
	bAck:= bAckP, 
	i_bConveyorOK:= i_bConveyor_3_Ok, 
	stStartEvent:= , 
	stRunEvent:= , 
	bMotorOn=> , 
	bError=> , 
	sError=> , 
	q_bConveyorOnL=> q_bConveyor_3, 
	q_bConveyorOnR=> , 
	q_bConveyorRst=> );

fbConveyor_4(
	sName:= 'Konveyor motor M4', 
	bEn:= i_bLO1_Main, 
	bEHA:= NOT bManualMode, 
	bDisableManualCmd:= NOT bManualMode, 
	bConveyorOnL:= , 
	bConveyorOnR:= , 
	timReset:= , 
	bAck:= bAckP, 
	i_bConveyorOK:= i_bConveyor_4_Ok, 
	stStartEvent:= , 
	stRunEvent:= , 
	bMotorOn=> , 
	bError=> , 
	sError=> , 
	q_bConveyorOnL=> q_bConveyor_4, 
	q_bConveyorOnR=> , 
	q_bConveyorRst=> );

fbConveyor_5(
	sName:= 'Konveyor motor M5', 
	bEn:= i_bLO1_Main, 
	bEHA:= NOT bManualMode, 
	bDisableManualCmd:= NOT bManualMode, 
	bConveyorOnL:= , 
	bConveyorOnR:= , 
	timReset:= , 
	bAck:= bAckP, 
	i_bConveyorOK:= i_bConveyor_5_Ok, 
	stStartEvent:= , 
	stRunEvent:= , 
	bMotorOn=> , 
	bError=> , 
	sError=> , 
	q_bConveyorOnL=> q_bConveyor_5, 
	q_bConveyorOnR=> , 
	q_bConveyorRst=> );

fbConveyor_6(
	sName:= 'Konveyor motor M6', 
	bEn:= i_bLO1_Main, 
	bEHA:= NOT bManualMode, 
	bDisableManualCmd:= NOT bManualMode, 
	bConveyorOnL:= , 
	bConveyorOnR:= , 
	timReset:= , 
	bAck:= bAckP, 
	i_bConveyorOK:= i_bConveyor_6_Ok, 
	stStartEvent:= , 
	stRunEvent:= , 
	bMotorOn=> , 
	bError=> , 
	sError=> , 
	q_bConveyorOnL=> q_bConveyor_6, 
	q_bConveyorOnR=> , 
	q_bConveyorRst=> );

fbConveyor_7(
	sName:= 'Konveyor motor M7', 
	bEn:= i_bLO1_Main, 
	bEHA:= NOT bManualMode, 
	bDisableManualCmd:= NOT bManualMode, 
	bConveyorOnL:= , 
	bConveyorOnR:= , 
	timReset:= , 
	bAck:= bAckP, 
	i_bConveyorOK:= i_bConveyor_7_Ok, 
	stStartEvent:= , 
	stRunEvent:= , 
	bMotorOn=> , 
	bError=> , 
	sError=> , 
	q_bConveyorOnL=> q_bConveyor_7, 
	q_bConveyorOnR=> , 
	q_bConveyorRst=> );

fbConveyor_8(
	sName:= 'Konveyor motor M8', 
	bEn:= i_bLO1_Main, 
	bEHA:= NOT bManualMode, 
	bDisableManualCmd:= NOT bManualMode, 
	bConveyorOnL:= , 
	bConveyorOnR:= , 
	timReset:= , 
	bAck:= bAckP, 
	i_bConveyorOK:= i_bConveyor_8_Ok, 
	stStartEvent:= , 
	stRunEvent:= , 
	bMotorOn=> , 
	bError=> , 
	sError=> , 
	q_bConveyorOnL=> q_bConveyor_8, 
	q_bConveyorOnR=> , 
	q_bConveyorRst=> );

fbConveyor_9(
	sName:= 'Konveyor motor M9', 
	bEn:= i_bLO1_Main, 
	bEHA:= NOT bManualMode, 
	bDisableManualCmd:= NOT bManualMode, 
	bConveyorOnL:= , 
	bConveyorOnR:= , 
	timReset:= , 
	bAck:= bAckP, 
	i_bConveyorOK:= i_bConveyor_9_Ok, 
	stStartEvent:= , 
	stRunEvent:= , 
	bMotorOn=> , 
	bError=> , 
	sError=> , 
	q_bConveyorOnL=> q_bConveyor_9, 
	q_bConveyorOnR=> , 
	q_bConveyorRst=> );

fbConveyor_10(
	sName:= 'Konveyor motor M10', 
	bEn:= i_bLO1_Main, 
	bEHA:= NOT bManualMode, 
	bDisableManualCmd:= NOT bManualMode, 
	bConveyorOnL:= , 
	bConveyorOnR:= , 
	timReset:= , 
	bAck:= bAckP, 
	i_bConveyorOK:= i_bConveyor_10_Ok, 
	stStartEvent:= , 
	stRunEvent:= , 
	bMotorOn=> , 
	bError=> , 
	sError=> , 
	q_bConveyorOnL=> q_bConveyor_10, 
	q_bConveyorOnR=> , 
	q_bConveyorRst=> );

fbConveyor_11(
	sName:= 'Konveyor motor M11', 
	bEn:= i_bLO1_Main, 
	bEHA:= NOT bManualMode, 
	bDisableManualCmd:= NOT bManualMode, 
	bConveyorOnL:= , 
	bConveyorOnR:= , 
	timReset:= , 
	bAck:= bAckP, 
	i_bConveyorOK:= i_bConveyor_11_Ok, 
	stStartEvent:= , 
	stRunEvent:= , 
	bMotorOn=> , 
	bError=> , 
	sError=> , 
	q_bConveyorOnL=> q_bConveyor_11, 
	q_bConveyorOnR=> , 
	q_bConveyorRst=> );
END_ACTION

ACTION Routers:
fbRouter_CNC1_puffer(
	bEnable:= i_bLO1_Main, 
	bErrorAck:= bAckP, 
	bManualMode:= bManualMode,
	bStepEnable:= bStepEnable, 
	stTagData:= fbRFID_Readers[7].Ch1_TagData, 
	bPaletteStopperIn:= fbS17.bPalletAtStopper, 
	bStopperReadyBase:= fbS3.bReady, 
	bStopperReadyWork:= fbS20.bReady, 
	nReqTarget:= 1, 					// CNC1 Puffer 	-> ST_Dut_Data
	nNextTarget:= 2,					// CNC1  		-> ST_Dut_Data
	fbRouter:= ADR(fbZ18),
	arrPaletteData:= ADR(arrPalette));

fbRouter_CNC2_puffer(
	bEnable:= i_bLO1_Main, 
	bErrorAck:= bAckP, 
	bManualMode:= bManualMode,
	bStepEnable:= bStepEnable, 
	stTagData:= fbRFID_Readers[6].Ch1_TagData, 
	bPaletteStopperIn:= fbS13.bPalletAtStopper, 
	bStopperReadyBase:= fbS5.bReady, 
	bStopperReadyWork:= fbS29.bReady, 
	nReqTarget:= 3, 					// CNC2 Puffer 	-> ST_Dut_Data
	nNextTarget:= 4,					// CNC2  		-> ST_Dut_Data
	fbRouter:= ADR(fbZ16),
	arrPaletteData:= ADR(arrPalette));

fbRouter_CNC3_puffer(
	bEnable:= i_bLO1_Main, 
	bErrorAck:= bAckP, 
	bManualMode:= bManualMode,
	bStepEnable:= bStepEnable, 
	stTagData:= fbRFID_Readers[5].Ch1_TagData, 
	bPaletteStopperIn:= fbS14.bPalletAtStopper, 
	bStopperReadyBase:= fbS8.bReady, 
	bStopperReadyWork:= fbS11.bReady, 
	nReqTarget:= 5, 					// CNC3 Puffer 	-> ST_Dut_Data
	nNextTarget:= 6,					// CNC3  		-> ST_Dut_Data
	fbRouter:= ADR(fbZ14),
	arrPaletteData:= ADR(arrPalette));
END_ACTION

ACTION Stoppers:
fbS24(			(*-----=== Kardex alsó pozíció 2. utáni torlasztás ===-----*)
	bNextReady:= fbS19.bReady, 
	bMotorRun:= i_bLO1_Main, 
	tToNextStopper:= T#5s, 
	bStationReady:= TRUE, 
	bStationFinished:= TRUE, 
	i_bPalettSensor:= GVL_ConveyorSystem.i_stSensorHub_2.Channel_5, 
	i_bPalettSensor2:= GVL_ConveyorSystem.i_stSensorHub_2.Channel_7, 
	q_bStopperDown=> GVL_ConveyorSystem.q_bS24);
	
fbS19(			(*-----=== Stopper kiemelő 1A előtt leválogatás ===-----*)
	bNextReady:= fbS1.bReady AND NOT fbS20.bPalletSent AND NOT((fbLift_1A.nState = 10000 OR fbLift_1B.nState = 10000)AND fbS20.i_bPalettSensor), 
	bMotorRun:= i_bLO1_Main, 
	tToNextStopper:= T#5s, 
	bStationReady:= TRUE, 
	bStationFinished:= TRUE, 
	i_bPalettSensor:= GVL_ConveyorSystem.i_stSensorHub_1.Channel_2,
	q_bStopperDown=> GVL_ConveyorSystem.q_bS19);

(****************************************************************************************)
(************************************** CNC1 ********************************************)
(****************************************************************************************)	
fbS1(			(*-----=== Stopper kiemelő 1A ===-----*)
	bNextReady:= fbS2.bReady, 
	bMotorRun:= i_bLO1_Main, 
	bStationReady:= fbLift_1A.nState = 10000 OR fbLift_1A.nState = 12000, 
	bStationFinished:= fbLift_1A.nState = 14000 OR fbLift_1A.nState = 12000, 
	i_bPalettSensor:= GVL_ConveyorSystem.i_stSensorHub_7.Channel_6, 
	q_bStopperDown=> GVL_ConveyorSystem.q_bS1);
	
fbS2(			(*-----=== Stopper kiemelő 1B ===-----*)
	bNextReady:= fbS17.bReady, 
	bMotorRun:= i_bLO1_Main, 
	bStationReady:= fbLift_1B.nState = 10000 OR fbLift_1B.nState = 12000, 
	bStationFinished:= fbLift_1B.nState = 14000 OR fbLift_1B.nState = 12000, 
	i_bPalettSensor:= GVL_ConveyorSystem.i_stSensorHub_6.Channel_6,
	q_bStopperDown=> GVL_ConveyorSystem.q_bS2);
	
fbS17(			(*-----=== CNC1 Puffer, Stopper kiemelő 1B után===-----*)
	bNextReady:= fbS3.bReady AND NOT fbS16.bPalletSent AND NOT((fbLift_2A.nState = 10000 OR fbLift_2B.nState = 10000)AND fbS16.i_bPalettSensor), 
	bMotorRun:= i_bLO1_Main, 
	tToNextStopper:= T#5s, 
	bStationReady:= fbRouter_CNC1_puffer.nState = 10000, 
	bStationFinished:= fbRouter_CNC1_puffer.nState = 12000 OR fbRouter_CNC1_puffer.nState = 13000, 
	i_bPalettSensor:= GVL_ConveyorSystem.i_stSensorHub_5.Channel_4, 
	q_bStopperDown=> GVL_ConveyorSystem.q_bS17);

fbS20(			(*-----=== CNC1 Puffer küldés ===-----*)
	bNextReady:= fbS1.bReady AND NOT fbS19.bPalletSent, 
	bMotorRun:= i_bLO1_Main, 
	tToNextStopper:= T#5s, 
	bStationReady:= TRUE, 
	bStationFinished:=  TRUE, 
	i_bPalettSensor:= GVL_ConveyorSystem.i_stSensorHub_5.Channel_6, 
	i_bPalettSensor2:= GVL_ConveyorSystem.i_stSensorHub_4.Channel_3,  
	q_bStopperDown=> GVL_ConveyorSystem.q_bS20);

(****************************************************************************************)
(************************************** CNC2 ********************************************)
(****************************************************************************************)	
fbS3(			(*-----=== Stopper kiemelő 2A ===-----*)
	bNextReady:= fbS4.bReady, 
	bMotorRun:= i_bLO1_Main, 
	bStationReady:= fbLift_2A.nState = 10000 OR fbLift_2A.nState = 12000, 
	bStationFinished:= fbLift_2A.nState = 14000 OR fbLift_2A.nState = 12000, 
	i_bPalettSensor:= GVL_ConveyorSystem.i_stSensorHub_10.Channel_6, 
	q_bStopperDown=> GVL_ConveyorSystem.q_bS3);	
	
fbS4(			(*-----=== Stopper kiemelő 2B ===-----*)
	bNextReady:= fbS13.bReady, 
	bMotorRun:= i_bLO1_Main, 
	bStationReady:= fbLift_2B.nState = 10000 OR fbLift_2B.nState = 12000, 
	bStationFinished:= fbLift_2B.nState = 14000 OR fbLift_2B.nState = 12000, 
	i_bPalettSensor:= GVL_ConveyorSystem.i_stSensorHub_11.Channel_6, 
	q_bStopperDown=> GVL_ConveyorSystem.q_bS4);

fbS13(			(*-----=== CNC2 Puffer, Stopper kiemelő 2B után===-----*)
	bNextReady:= fbS5.bReady AND NOT fbS11.bPalletSent AND NOT((fbLift_3A.nState = 10000 OR fbLift_3B.nState = 10000)AND fbS11.i_bPalettSensor), 
	bMotorRun:= i_bLO1_Main, 
	tToNextStopper:= T#5s, 
	bStationReady:= fbRouter_CNC2_puffer.nState = 10000, 
	bStationFinished:= fbRouter_CNC2_puffer.nState = 12000 OR fbRouter_CNC2_puffer.nState = 13000, 
	i_bPalettSensor:= GVL_ConveyorSystem.i_stSensorHub_8.Channel_4, 
	q_bStopperDown=> GVL_ConveyorSystem.q_bS13);

fbS16(			(*-----=== CNC2 Puffer küldés ===-----*)
	bNextReady:= fbS3.bReady, 
	bMotorRun:= i_bLO1_Main, 
	tToNextStopper:= T#5s, 
	tToNextStopper:= T#5s, 
	bStationReady:= fbZ17.bWorkPosStab, 
	bStationFinished:= fbZ17.bWorkPosStab, 
	i_bPalettSensor:= GVL_ConveyorSystem.i_stSensorHub_8.Channel_6, 
	i_bPalettSensor2:= GVL_ConveyorSystem.i_stSensorHub_12.Channel_2, 
	q_bStopperDown=> GVL_ConveyorSystem.q_bS16);


(****************************************************************************************)
(************************************** CNC3 ********************************************)
(****************************************************************************************)		
fbS5(			(*-----=== Stopper kiemelő 3A ===-----*)
	bNextReady:= fbS6.bReady, 
	bMotorRun:= i_bLO1_Main, 
	bStationReady:= fbLift_3A.nState = 10000 OR fbLift_3A.nState = 12000, 
	bStationFinished:= fbLift_3A.nState = 14000 OR fbLift_3A.nState = 12000, 
	i_bPalettSensor:= GVL_ConveyorSystem.i_stSensorHub_14.Channel_6, 
	q_bStopperDown=> GVL_ConveyorSystem.q_bS5);
	
fbS6(			(*-----=== Stopper kiemelő 3B ===-----*)
	bNextReady:= fbS11.bReady, 
	bMotorRun:= i_bLO1_Main, 
	bStationReady:= fbLift_3B.nState = 10000 OR fbLift_3B.nState = 12000, 
	bStationFinished:= fbLift_3B.nState = 14000 OR fbLift_3B.nState = 12000, 
	i_bPalettSensor:= GVL_ConveyorSystem.i_stSensorHub_15.Channel_6, 
	q_bStopperDown=> GVL_ConveyorSystem.q_bS6);

fbS14(
	bNextReady:= fbS8.bReady, 
	bMotorRun:= i_bLO1_Main, 
	tToNextStopper:= T#5s, 
	bStationReady:= fbRouter_CNC3_puffer.nState = 10000, 
	bStationFinished:= fbRouter_CNC3_puffer.nState = 12000 OR fbRouter_CNC3_puffer.nState = 13000, 
	i_bPalettSensor:= GVL_ConveyorSystem.i_stSensorHub_13.Channel_5, 
	q_bStopperDown=> GVL_ConveyorSystem.q_bS14);

fbS11(			(*-----=== CNC3 Puffer küldés ===-----*)
	bNextReady:= fbS5.bReady, 
	bMotorRun:= i_bLO1_Main, 
	tToNextStopper:= T#5s, 
	bStationReady:= TRUE,  
	bStationFinished:= , 
	i_bPalettSensor:= GVL_ConveyorSystem.i_stSensorHub_13.Channel_2, 
	i_bPalettSensor2:= GVL_ConveyorSystem.i_stSensorHub_13.Channel_4, 
	q_bStopperDown=> GVL_ConveyorSystem.q_bS11);

(****************************************************************************************)
(*********************** Alsó konvejor visszahordás *************************************)
(****************************************************************************************)
fbS8(			(*-----=== alsó visszahordó 1. torlasztás ===-----*)
	bNextReady:= fbS27.bReady, 
	bMotorRun:= i_bLO1_Main, 
	tToNextStopper:= T#5S, 
	bStationReady:= TRUE, 
	bStationFinished:= TRUE, 
	i_bPalettSensor:= GVL_ConveyorSystem.i_stSensorHub_9.Channel_6, 
	i_bPalettSensor2:= GVL_ConveyorSystem.i_stSensorHub_9.Channel_3, 
	q_bStopperDown=> GVL_ConveyorSystem.q_bS8);

fbS27(			(*-----=== alsó visszahordó 2. torlasztás ===-----*)
	bNextReady:= fbS21.bReady, 
	bMotorRun:= i_bLO1_Main, 
	tToNextStopper:= T#5S, 
	bStationReady:= TRUE, 
	bStationFinished:= TRUE, 
	i_bPalettSensor:= GVL_ConveyorSystem.i_stSensorHub_3.Channel_6, 
	i_bPalettSensor2:= GVL_ConveyorSystem.i_stSensorHub_4.Channel_0, 
	q_bStopperDown=> GVL_ConveyorSystem.q_bS27);

fbS29(			(*-----=== alsó visszahordó S19 után 2nd felfogás ===-----*)
	bNextReady:= , 
	bMotorRun:= i_bLO1_Main, 
	tToNextStopper:= T#5S, 
	bStationReady:= TRUE, 
	bStationFinished:= TRUE, 
	i_bPalettSensor:= GVL_ConveyorSystem.i_stSensorHub_0.Channel_1, 
	q_bStopperDown=> GVL_ConveyorSystem.q_bS29);

fbS21(			(*-----=== alsó visszahordó 3. torlasztás ===-----*)
	bNextReady:= fbS22.bReady, 
	bMotorRun:= i_bLO1_Main, 
	tToNextStopper:= T#5S, 
	bStationReady:= TRUE, 
	bStationFinished:= TRUE, 
	i_bPalettSensor:= GVL_ConveyorSystem.i_stSensorHub_1.Channel_6, 
	i_bPalettSensor2:= GVL_ConveyorSystem.i_stSensorHub_2.Channel_0, 
	q_bStopperDown=> GVL_ConveyorSystem.q_bS21);
	
fbS22(			(*-----=== Kardex alsó pozíció 1. ===-----*)
	bNextReady:= fbS23.bReady, 
	bMotorRun:= i_bLO1_Main, 
	tToNextStopper:= T#5S, 
	bStationReady:= TRUE, 
	bStationFinished:= TRUE, 
	i_bPalettSensor:= GVL_ConveyorSystem.i_stSensorHub_2.Channel_1, 
	q_bStopperDown=> GVL_ConveyorSystem.q_bS22);
	
fbS23(			(*-----=== Kardex alsó pozíció 2. ===-----*)
	bNextReady:= fbS24.bReady, 
	bMotorRun:= i_bLO1_Main, 
	tToNextStopper:= T#5S, 
	bStationReady:= NOT RobotKardexProgram.fbRobot.RobotIn.Status.bRobotInStrip_3 AND NOT RobotKardexProgram.bInterlock_Strip3, 
	bStationFinished:= NOT RobotKardexProgram.fbRobot.RobotIn.Status.bRobotInStrip_3 AND NOT RobotKardexProgram.bInterlock_Strip3, 
	i_bPalettSensor:= GVL_ConveyorSystem.i_stSensorHub_2.Channel_3, 
	q_bStopperDown=> GVL_ConveyorSystem.q_bS23);
	
(****************************************************************************************)
(************************** Felső konvejor behordás *************************************)
(****************************************************************************************)
fbS7(			(*-----=== Operátori pozíció ===-----*)
	bNextReady:= fbS10.bReady, 
	bMotorRun:= i_bLO1_Main, 
	tToNextStopper:= T#1s, 
	bStationReady:= UploadingProgram.nState = 10000, 
	bStationFinished:= UploadingProgram.nState = 12000, 
	i_bPalettSensor:= GVL_ConveyorSystem.i_stSensorHub_17.Channel_0, 
	q_bStopperDown=> GVL_ConveyorSystem.q_bS7);
	
fbS10(
	bNextReady:= fbS9.bReady, 
	bMotorRun:= i_bLO1_Main, 
	tToNextStopper:= T#5s, 
	bStationReady:= TRUE,  
	bStationFinished:= TRUE, 
	i_bPalettSensor:= GVL_ConveyorSystem.i_stSensorHub_17.Channel_5, 
	i_bPalettSensor2:= GVL_ConveyorSystem.i_stSensorHub_17.Channel_7, 
	q_bStopperDown=> GVL_ConveyorSystem.q_bS10);

fbS9(
	bNextReady:= fbS18.bReady, 
	bMotorRun:= i_bLO1_Main, 
	tToNextStopper:= T#5s, 
	bStationReady:= TRUE, 
	bStationFinished:= TRUE, 
	i_bPalettSensor:= GVL_ConveyorSystem.i_stSensorHub_16.Channel_0, 
	i_bPalettSensor2:= GVL_ConveyorSystem.i_stSensorHub_16.Channel_2, 
	q_bStopperDown=> GVL_ConveyorSystem.q_bS9);

fbS18(
	bNextReady:= fbS15.bReady, 
	bMotorRun:= i_bLO1_Main, 
	tToNextStopper:= T#15s, 
	bStationReady:= TRUE,  
	bStationFinished:= TRUE, 
	i_bPalettSensor:= GVL_ConveyorSystem.i_stSensorHub_12.Channel_5, 
	i_bPalettSensor2:= GVL_ConveyorSystem.i_stSensorHub_12.Channel_7, 
	q_bStopperDown=> GVL_ConveyorSystem.q_bS18);

fbS15(
	bNextReady:= fbS26.bReady, 
	bMotorRun:= i_bLO1_Main, 
	tToNextStopper:= T#15s, 
	bStationReady:= TRUE,  
	bStationFinished:= TRUE, 
	i_bPalettSensor:= GVL_ConveyorSystem.i_stSensorHub_12.Channel_3, 
	i_bPalettSensor2:= GVL_ConveyorSystem.i_stSensorHub_9.Channel_4, 
	q_bStopperDown=> GVL_ConveyorSystem.q_bS15);
	
fbS26(
	bNextReady:= fbS25.bReady, 
	bMotorRun:= i_bLO1_Main, 
	tToNextStopper:= T#15s, 
	bStationReady:= TRUE,  
	bStationFinished:= TRUE, 
	i_bPalettSensor:= GVL_ConveyorSystem.i_stSensorHub_0.Channel_3, 
	i_bPalettSensor2:= GVL_ConveyorSystem.i_stSensorHub_4.Channel_4,  
	q_bStopperDown=> GVL_ConveyorSystem.q_bS26);

fbS25(
	bNextReady:= fbS32.bReady, 
	bMotorRun:= i_bLO1_Main, 
	tToNextStopper:= T#5s, 
	bStationReady:= TRUE, 
	bStationFinished:= TRUE, 
	i_bPalettSensor:= GVL_ConveyorSystem.i_stSensorHub_3.Channel_2, 
	i_bPalettSensor2:= GVL_ConveyorSystem.i_stSensorHub_0.Channel_0,  
	q_bStopperDown=> GVL_ConveyorSystem.q_bS25);
	
fbS32(
	bNextReady:= FALSE, 
	bMotorRun:= i_bLO1_Main, 
	tToNextStopper:= T#1s, 
	bStationReady:= NOT RobotKardexProgram.fbRobot.RobotIn.Status.bRobotInStrip_1 AND NOT RobotKardexProgram.bInterlock_Strip1, 
	bStationFinished:= NOT RobotKardexProgram.fbRobot.RobotIn.Status.bRobotInStrip_1 AND NOT RobotKardexProgram.bInterlock_Strip1, 
	i_bPalettSensor:= GVL_ConveyorSystem.i_stSensorHub_3.Channel_0, 
	q_bStopperDown=> GVL_ConveyorSystem.q_bS32);

(****************************************************************************************)
(************************** Felső konvejor kihordás *************************************)
(****************************************************************************************)
fbS30(
	bNextReady:= fbS31.bReady, 
	bMotorRun:= i_bLO1_Main, 
	tToNextStopper:= T#10s, 
	bStationReady:= TRUE, 
	bStationFinished:= TRUE, 
	i_bPalettSensor:= GVL_ConveyorSystem.i_stSensorHub_4.Channel_1, 
	i_bPalettSensor2:= GVL_ConveyorSystem.i_stSensorHub_4.Channel_5,  
	q_bStopperDown=> GVL_ConveyorSystem.q_bS30);	

fbS31(
	bNextReady:= fbS12.bReady, 
	bMotorRun:= i_bLO1_Main, 
	tToNextStopper:= T#10s, 
	bStationReady:= TRUE, 
	bStationFinished:= TRUE, 
	i_bPalettSensor:= GVL_ConveyorSystem.i_stSensorHub_9.Channel_2, 
	i_bPalettSensor2:= GVL_ConveyorSystem.i_stSensorHub_9.Channel_5,  
	q_bStopperDown=> GVL_ConveyorSystem.q_bS31);	

fbS12(
	bNextReady:= fbS28.bReady, 
	bMotorRun:= i_bLO1_Main, 
	tToNextStopper:= T#15s, 
	bStationReady:= TRUE, 
	bStationFinished:= TRUE, 
	i_bPalettSensor:= GVL_ConveyorSystem.i_stSensorHub_16.Channel_5, 
	i_bPalettSensor2:= GVL_ConveyorSystem.i_stSensorHub_9.Channel_0,  
	q_bStopperDown=> GVL_ConveyorSystem.q_bS12);

fbS28(			(*-----=== Operátori pozíció Fix nincs vezérelve ===-----*)
	bNextReady:= FALSE, 
	bMotorRun:= i_bLO1_Main, 
	bStationReady:= TRUE,			// Satuzó állomás paletta kérése 
	bStationFinished:= TRUE, 
	i_bPalettSensor:= GVL_ConveyorSystem.i_stSensorHub_17.Channel_2, 
	q_bStopperDown=> );
END_ACTION

END_PROGRAM

// ---- POUs/UploadingStation/UploadingProgram.TcPOU
PROGRAM UploadingProgram
VAR	(* Control *)
	nState						: UDINT;
	nStatePrevious				: UDINT;
	sState						: STRING(500);
	bError						: BOOL;
	fbCycleTime					: TON;
	nCycleTime					: REAL;
END_VAR

VAR CONSTANT
	iLastStatesMax				: INT := 500;
END_VAR
VAR //LastStates
	anLastStates				:ARRAY[0..iLastStatesMax] OF UDINT;
    iLastStates					:INT;
END_VAR
VAR (* Operator *)
	arRobotEvents				: ARRAY [0..15] OF TcEventEntry;
END_VAR
VAR (* Test variables *)
	stTagData					: ST_Tag_Data;
	PaletteId					: INT;
	tRFID_Timeout				: TON;
	nLastTarget					: UINT := 5;
END_VAR
VAR // MySQL
	
END_VAR

MySQL();
stTagData := GVL_RFID.fbRFID_Readers[4].Ch1_TagData;

(*Error handling*)
IF nState > 0 AND nState < 150000 THEN
	nStatePrevious := nState;
END_IF

(*Maintance*)
IF bManualMode THEN
	nState := 150000;
END_IF

(*Emergency*)
IF NOT i_bLO1_Main THEN
	nState := 0;
END_IF

(*Last states*)
IF(nState >= 1000) AND (nState < 150000) THEN
(*Steps before any state*)
	IF anLastStates[0] <> nState THEN
		FOR iLastStates:=iLastStatesMax TO 1 BY -1 DO
			anLastStates[iLastStates]:= anLastStates[iLastStates-1];
		END_FOR
		anLastStates[0]:= nState;
	END_IF
END_IF	

IF FALSE
THEN
	bError  :=  TRUE;
END_IF



CASE nState OF
{region "Alaphelyzet felvétel"}
	(****************************************************************************************)
	(******************************* Alaphelyzetfelvétel ************************************)
	(****************************************************************************************)	
	0:		(*-----=== Kimenetek törlése ===-----*)
		sState := CONCAT(UDINT_TO_STRING(nState) ,' - A biztonsági kör nem aktív');
		
		IF i_bLO1_Main AND NOT bManualMode THEN
			nState := nState + 20;
		END_IF
	20:
		nState := 10000;
{endregion}
		
{region "Alaphelyzet"}
	(****************************************************************************************)
	(*********************************** Alaphelyzet ****************************************)
	(****************************************************************************************)	
	10000:		(* -----=== Várakozás parancsra ===----- *)
		sState := CONCAT(UDINT_TO_STRING(nState) ,' - Alaphelyzet');
		IF fbS7.bPalletAtStopper THEN
			nState := 11000;
		END_IF
{endregion}

{region "Alaphelyzet"}
	(****************************************************************************************)
	(*********************************** Paletta fogadása ***********************************)
	(****************************************************************************************)	
	11000:		(*-----=== RFID ellenőrzése ===-----*)
		sState := CONCAT(UDINT_TO_STRING(nState) ,' - RFID ellenőrzés');
		IF stTagData.Status <> E_TagStatus.NotPresent THEN
			IF stTagData.Code > 0 AND stTagData.Code <= 100 THEN
				IF bStepEnable THEN
					PaletteId := ULINT_TO_INT(stTagData.Code);
					nState := nState + 20;							// -> Valid RFID adat
				END_IF
			END_IF
		ELSIF tRFID_Timeout.Q THEN
			nState := 14000;										// -> RFID hiba -> tovább küldés
		END_IF

	11020:		(*-----=== Paletta adat feltöltés ===-----*)
		sState := CONCAT(UDINT_TO_STRING(nState) ,' - Paletta adat feltöltés');
		nLastTarget := nLastTarget + 2;
		IF nLastTarget > 5 THEN
			nLastTarget := 1;
		END_IF
		GVL_Palette.arrPalette[PaletteId].nDutId := 1;
		GVL_Palette.arrPalette[PaletteId].sSerNr := 'VM001234';
		GVL_Palette.arrPalette[PaletteId].nPaletteId := PaletteId;
		GVL_Palette.arrPalette[PaletteId].nCamFileId := 0;
		GVL_Palette.arrPalette[PaletteId].nDimX := 40;
		GVL_Palette.arrPalette[PaletteId].nDimY := 45;
		GVL_Palette.arrPalette[PaletteId].nDimZ := 30;
		GVL_Palette.arrPalette[PaletteId].nPosX := 0;
		GVL_Palette.arrPalette[PaletteId].nPosX := 0;
		GVL_Palette.arrPalette[PaletteId].nTorque := 35;
		GVL_Palette.arrPalette[PaletteId].nWeight := 200;
		GVL_Palette.arrPalette[PaletteId].bPass := TRUE;
		GVL_Palette.arrPalette[PaletteId].bDutInVise := FALSE;
		GVL_Palette.arrPalette[PaletteId].bDone := FALSE;
		GVL_Palette.arrPalette[PaletteId].nState := 1;
		GVL_Palette.arrPalette[PaletteId].nTarget := nLastTarget;
		nState := nState + 20;

	11040:		(*-----=== Várakozás paletta indításra ===-----*)
		sState := CONCAT(UDINT_TO_STRING(nState) ,' - Várakozás paletta indításra');
		IF i_bCaptron THEN
			IF bStepEnable THEN
				nState := 12000;
			END_IF
		END_IF

	12000:		(*-----=== Várakozás paletta elengedésre ===-----*)
		sState := CONCAT(UDINT_TO_STRING(nState) ,' - Várakozás paletta indításra');
		IF NOT fbS7.bPalletAtStopper THEN
			IF bStepEnable THEN
				nState := nState + 20;
			END_IF
		END_IF
	
	12020:
		nState := 10000;
{endregion}
	
	150000: (* Maintenance *)
		sState := CONCAT(UDINT_TO_STRING(nState) ,' - Maintenance');
		IF NOT bManualMode THEN
			nState := 0;
		END_IF
		
	200000:(* Error handling *)
		sState := CONCAT(UDINT_TO_STRING(nState) ,CONCAT(' - Error, from this state: ' , sState));
		nState := 200020;
	
	200020:(* Error handling *)
		IF bAckP THEN
			CASE nStatePrevious OF
				0..9999: nState := 0;
//				10000..25000: nState := 10000;
//				30000..31000: nState := 30000;
			ELSE nState := 0;
			END_CASE
		END_IF	
		
	ELSE //Not a real step, for test purposes
		sState := CONCAT(UDINT_TO_STRING(nState) ,' - Not a real step, for test purposes');
END_CASE

(*Timers***************************************************)
fbCycleTime(IN:= nState > 10000 AND nState <= 95000, PT:= T#1D, Q=> , ET=> );
IF nState > 10000 AND nState <= 95000 THEN
	nCycleTime := TIME_TO_REAL(fbCycleTime.ET)/1000;
END_IF

tRFID_Timeout(IN:= fbS7.bPalletAtStopper AND stTagData.Status = E_TagStatus.NotPresent, PT:= T#2s, Q=> , ET=> );

(*Captron***************************************************)
IF nState = 11040 THEN
	q_bCaptronLED := bBL500p500;
ELSE
	q_bCaptronLED := FALSE;
END_IF

ACTION MySQL:
;
END_ACTION

END_PROGRAM

// ---- POUs/SQL_Test.TcPOU
PROGRAM SQL_Test
VAR
//	fbGetNextVise			: FB_SP_spGetNextVise;
END_VAR

//fbGetNextVise(
//	CncNumber:= , 
//	nRecordStartIndex:= 0, 
//	tTimeout:= , 
//	bExecute:= , 
//	bBusy=> , 
//	bError=> , 
//	ipResult=> , 
//	nViseNr=> );

END_PROGRAM

// ---- POUs/FBs/Pneumatics/FB_Stopper.TcPOU
FUNCTION_BLOCK FB_Stopper
VAR_INPUT
	sName				:STRING;
	bNextReady			:BOOL;				(* Következő stopper fogadókész *)
	bMotorRun			:BOOL;				(* Pályamotor jár *)
	tToNextStopper		:TIME := T#5S;		(* Ennél sűrűbben nem engedhet ki palettát *)
	bStationReady		:BOOL;				(* Állomás fogadókész/kiemelő lent van(ha van a stopperhez) *)
	bStationFinished	:BOOL;				(* Állomás kész, mehet a paletta(ha van a stopperhez) *)
	tPalletInStab		:TIME := T#50MS;	(* A stoppernél stabilan van paletta *)
	tPalletOutStab		:TIME := T#50MS;	(* A stoppernél stabilan nincs paletta *)
	i_bPalettSensor		AT %I* :BOOL;		(* Paletta érzékelő*)
END_VAR
VAR_OUTPUT
	bReady				:BOOL;
	bPalletAtStopper	:BOOL;
	bPalletSent			:BOOL;				(* Paletta küldés folyamatban/bekapcsolás *)
	q_bStopperDown		AT %Q* :BOOL;
END_VAR
VAR_IN_OUT
END_VAR
VAR
	tPalettOut			:TIME := T#100MS; (*Paletta kiengedéshez *)
	fbToNextStopper		:TON;
	fbPalettOut			:TON;
	fbEmpty				:TON;
	fbPalletInStab		:TON;
	fbPalletOutStab		:TON;
END_VAR

(*	Dokumentáció
	--------------------------------------------------------------------------------
	Leírás		:	Funkció blokk stopperekhez. 
	Név			:	FB_Stopper
	Módosító	:	Gyarmati Péter
	Dátum		:	2020.07.31
	Revízió		:	1.3
	--------------------------------------------------------------------------------
	Feltételek	:	-
	Változók	:	-
	Visu		:	-
	UserControl	:	-
	--------------------------------------------------------------------------------
	Részletek	:	-
	--------------------------------------------------------------------------------
	Használat	:	Allomas_nelkuli_stopper(
					bNextReady:= Stopper_allomassal.bReady, 
					bMotorRun:= i_bEMYOK, 
					bStationReady:= TRUE, 
					bStationFinished:= TRUE);
	
					Stopper_allomassal(
						bNextReady:= Kovistopper.bReady, 
						bMotorRun:= i_bEMYOK, 
						bStationReady:= nState = 10000, //ha ki van emelve a paletta, a bStationReady-t vegyük el, hogy ne engedjen rá még újat, itt csak alaphelyzetben jöhet
						bStationFinished:= nState = 95020 //ebben a státuszban az állomás végzett, paletta elengedésre vár);
*)

fbToNextStopper(IN:= bMotorRun AND NOT q_bStopperDown, PT:= tToNextStopper, Q=> );
fbPalettOut(IN:= q_bStopperDown AND NOT i_bPalettSensor AND bMotorRun, PT:= tPalettOut);
fbEmpty(IN:= NOT i_bPalettSensor AND NOT q_bStopperDown AND bMotorRun AND bStationReady, PT:= T#1S, Q=> bReady);			// PT:= T#3S eredetileg

fbPalletInStab(IN:= i_bPalettSensor AND bMotorRun, PT:= tPalletInStab);
fbPalletOutStab(IN:= NOT i_bPalettSensor AND NOT q_bStopperDown AND bMotorRun, PT:= tPalletOutStab);
IF fbPalletInStab.Q THEN
	bPalletAtStopper := TRUE;
END_IF
IF fbPalletOutStab.Q THEN
	bPalletAtStopper := FALSE;
END_IF

(*Paletta továbbengedés*)
IF bNextReady AND fbToNextStopper.Q AND i_bPalettSensor AND bMotorRun AND bStationFinished THEN
	q_bStopperDown := TRUE;
END_IF

IF fbPalettOut.Q THEN 
	q_bStopperDown := FALSE;
END_IF
bPalletSent := NOT fbToNextStopper.Q;

END_FUNCTION_BLOCK

// ---- POUs/FBs/Pneumatics/FB_Stopper2.TcPOU
FUNCTION_BLOCK FB_Stopper2
VAR_INPUT
	sName				:STRING;
	bNextReady			:BOOL;			(*Következő stopper fogadókész*)
	bMotorRun			:BOOL;			(*Pályamotor jár*)
	tToNextStopper		:TIME := T#5S;	(*Ennél sűrűbben nem engedhet ki palettát*)
	bStationReady		:BOOL;			(*Állomás fogadókész/kiemelő lent van(ha van a stopperhez)*)
	bStationFinished	:BOOL;			(*Állomás kész, mehet a paletta(ha van a stopperhez)*)
	i_bPalettSensor		AT %I* :BOOL;	(*Paletta érzékelő*)
	i_bPalettSensor2	AT %I* :BOOL;	(*Paletta érzékelő torlasztási maximum*)
END_VAR
VAR_OUTPUT
	bReady				:BOOL;
	bPalletSent			:BOOL;				(* Paletta küldés folyamatban/bekapcsolás *)
	q_bStopperDown		AT %Q* :BOOL;
END_VAR
VAR_IN_OUT
END_VAR
VAR
	tPalettOut			:TIME := T#100MS;	(*Paletta kiengedéshez *)
	fbToNextStopper		:TON;
	fbPalettOut			:TON;
	fbEmpty				:TON;
END_VAR

(*	Dokumentáció
	--------------------------------------------------------------------------------
	Leírás		:	Funkció blokk stopperekhez telítettség érzékelővel. 
	Név			:	FB_Stopper2
	Módosító	:	Gyarmati Péter
	Dátum		:	2020.07.31
	Revízió		:	1.3
	--------------------------------------------------------------------------------
	Feltételek	:	-
	Változók	:	-
	Visu		:	-
	UserControl	:	-
	--------------------------------------------------------------------------------
	Részletek	:	-
	--------------------------------------------------------------------------------
	Használat	:	Allomas_nelkuli_stopper(
					bNextReady:= Stopper_allomassal.bReady, 
					bMotorRun:= i_bEMYOK, 
					bStationReady:= TRUE, 
					bStationFinished:= TRUE);
	
					Stopper_allomassal(
						bNextReady:= Kovistopper.bReady, 
						bMotorRun:= i_bEMYOK, 
						bStationReady:= nState = 10000, //ha ki van emelve a paletta, a bStationReady-t vegyük el, hogy ne engedjen rá még újat, itt csak alaphelyzetben jöhet
						bStationFinished:= nState = 95020 //ebben a státuszban az állomás végzett, paletta elengedésre vár);
*)

fbToNextStopper(IN:= bMotorRun AND NOT q_bStopperDown, PT:= tToNextStopper, Q=>);
fbPalettOut(IN:= q_bStopperDown AND NOT i_bPalettSensor AND bMotorRun, PT:= tPalettOut);
fbEmpty(IN:= NOT i_bPalettSensor2 AND NOT q_bStopperDown AND bMotorRun AND bStationReady, PT:= T#1S, Q=> bReady);			// PT:= T#3S eredetileg

(*Paletta továbbengedés*)
IF bNextReady AND fbToNextStopper.Q AND i_bPalettSensor AND bMotorRun AND bStationFinished THEN
	q_bStopperDown := TRUE;
END_IF

IF fbPalettOut.Q THEN 
	q_bStopperDown := FALSE;
END_IF
bPalletSent := NOT fbToNextStopper.Q;

END_FUNCTION_BLOCK

// ---- POUs/FBs/FB_Conveyor.TcPOU
FUNCTION_BLOCK FB_Conveyor
VAR_INPUT
	sName					:STRING;
	bEn						:BOOL;				(*Enable - Engedély jel*)
	bEHA					:BOOL; 				(*Error-handling active - Hibafigyelés aktív*)
	bDisableManualCmd		:BOOL;				(*Manual control disable*)
	bConveyorOnL			:BOOL;				(*Control to Motor on - vezérlés parancs motor indításhoz*)
	bConveyorOnR			:BOOL;				(*Control to Motor on - vezérlés parancs motor indításhoz*)
	timReset				:TIME := T#2S;		(*Resettime - Hibatörlési idő*)
	bAck					:BOOL; 				(*Acknowledge - Hibanyugta*)
	i_bConveyorOK	AT %I*	:BOOL;				(*Conveyor drive OK - motorindító üzemkész*)
	stStartEvent			:TcEventEntry;		(*Event definition*)
	stRunEvent				:TcEventEntry;		(*Event definition*)
END_VAR
VAR_OUTPUT
	bMotorOn				:BOOL;				(* Motor on - Motor bekapcsolva *)
	bError					:BOOL;				(* Error bit - Hiba van *)
	sError					:STRING(255);		(* Error string - Hiba string *)
	q_bConveyorOnL	AT %Q*	:BOOL;				(* Motor on signal - Motor vezérlés bekapcsolása*)
	q_bConveyorOnR	AT %Q*	:BOOL;				(* Motor on signal - Motor vezérlés bekapcsolása*)
	q_bConveyorRst	AT %Q*	:BOOL;				(* Motor reset signal - Motor hibatörlés*)
END_VAR
VAR
	tMotorOn			:TON;
	tError,tFault		:TON;
	tReset				:TON;
	bErrOn,bErrRun		:BOOL;
	aErrorDesc			:ARRAY [0..1] OF STRING := [
	' motor hiba : a motorvezérlő nem indítható ', 
	' motor hiba : a motorvezérlő hibába van '];
	sEmpty				:STRING:='';
	bIsInitalized		:BOOL;
	fbStartAlarm		:FB_TcAlarm;
	fbRunAlarm			:FB_TcAlarm;
END_VAR

(*Hibanyugta*)
IF bAck OR NOT(bEHA) THEN
	bErrOn:=FALSE;
	bErrRun:=FALSE;
END_IF;

(* Motor bekapcsolási hiba *)
IF bEn AND bEHA AND (q_bConveyorOnL OR q_bConveyorOnR) AND NOT i_bConveyorOK THEN
	bErrOn:=TRUE;
	IF (fbStartAlarm.eConfirmationState <> 2 AND fbStartAlarm.nTimeCleared <> 0 AND fbStartAlarm.nTimeConfirmed <> 0) OR //Ha már volt alarm, akkor van bennük érték
		(fbStartAlarm.eConfirmationState = 1 AND fbStartAlarm.nTimeCleared = 0 AND fbStartAlarm.nTimeConfirmed = 0)	//Első futás esetén
	THEN
		fbStartAlarm.Raise(0);
	END_IF
END_IF;

(* Motor üzemzavar *)
tFault(IN:= bEn AND bEHA AND NOT i_bConveyorOK AND NOT bErrRun, PT:= T#5S);
IF tFault.Q THEN
	bErrRun:=TRUE;
	IF (fbRunAlarm.eConfirmationState <> 2 AND fbRunAlarm.nTimeCleared <> 0 AND fbRunAlarm.nTimeConfirmed <> 0) OR //Ha már volt alarm, akkor van bennük érték
		(fbRunAlarm.eConfirmationState = 1 AND fbRunAlarm.nTimeCleared = 0 AND fbRunAlarm.nTimeConfirmed = 0)	//Első futás esetén
	THEN
		fbRunAlarm.Raise(0);
	END_IF
END_IF;

(* Hibagyűjtő *)
bError := bErrOn OR bErrRun;

(*Vezérlés*)
IF 		bEn AND bConveyorOnL AND NOT bConveyorOnR AND i_bConveyorOK AND (NOT(bEHA) OR NOT(bError)) THEN
			q_bConveyorOnL := TRUE;
			q_bConveyorOnR := FALSE;
ELSIF	bEn AND NOT bConveyorOnL AND bConveyorOnR AND i_bConveyorOK AND (NOT(bEHA) OR NOT(bError)) THEN
			q_bConveyorOnL := FALSE;
			q_bConveyorOnR := TRUE;
ELSE
	q_bConveyorOnL := FALSE;
	q_bConveyorOnR := FALSE;
END_IF

(* Motor bekapcsolva *)
tMotorOn(IN:= (q_bConveyorOnL OR q_bConveyorOnR) AND NOT bError, 
	PT:= T#1S,
	Q=>  bMotorOn);

(* Manual reset *)
IF bError AND bAck AND NOT q_bConveyorRst THEN
	q_bConveyorRst := TRUE;
END_IF

tReset(IN:= q_bConveyorRst, PT:= timReset, Q=> , ET=> );
IF tReset.Q THEN
	q_bConveyorRst := FALSE;
END_IF

(*Hiba string*)
IF bErrOn OR bErrRun THEN
	sError := sName;
	IF bErrOn THEN
		sError :=  CONCAT(sError, aErrorDesc[0]);
	END_IF
	IF bErrRun THEN
		sError :=  CONCAT(sError, aErrorDesc[1]);
	END_IF
ELSE
	sError := sEmpty;
END_IF

(*Hiba kezelés Tc3_EventLogger*)
IF NOT bIsInitalized THEN
	bIsInitalized := TRUE;
	fbStartAlarm.CreateEx(stStartEvent, TRUE, 0);
	fbRunAlarm.CreateEx(stRunEvent, TRUE, 0);
END_IF

(*Hiba törlés (nyugtázott és megszűnt)*)
IF fbStartAlarm.eConfirmationState = 3 AND NOT bError THEN
	fbStartAlarm.Clear(0, FALSE);
END_IF	
IF fbRunAlarm.eConfirmationState = 3 AND NOT bError THEN
	fbRunAlarm.Clear(0, FALSE);
END_IF

END_FUNCTION_BLOCK

// ---- POUs/FBs/Lift/FB_Lift.TcPOU
FUNCTION_BLOCK FB_Lift
VAR_INPUT
	bEnable					: BOOL;
	bErrorAck				: BOOL;
	bManualMode				: BOOL;
	bStepEnable				: BOOL;
	bBeforeStopperSent		: BOOL;
	stTagData				: ST_Tag_Data;
	nReqTarget				: UINT;
END_VAR
VAR_INPUT
	fbLift					: POINTER TO FB_Bistabil;
	fbLock					: POINTER TO FB_Bistabil;
	fbStopper				: POINTER TO FB_Stopper;
	arrPaletteData			: POINTER TO ARRAY [0..200] OF ST_Dut_Data;
END_VAR
VAR_OUTPUT
	nTagID					: ULINT;
	bPalletAtStopper		: BOOL;
END_VAR
VAR	(* Control *)
	nState						: UDINT;
	nStatePrevious				: UDINT;
	sState						: STRING(500);
	fbCycleTime					: TON;
	nCycleTime					: REAL;
	bError						: BOOL;
	tRFID_Timeout				: TON;
END_VAR
VAR CONSTANT
	iLastStatesMax				: INT := 500;
END_VAR
VAR (* LastStates *)
	anLastStates				: ARRAY[0..iLastStatesMax] OF UDINT;
    iLastStates					: INT;
END_VAR

(*Error handling*)
IF nState > 0 AND nState < 150000 THEN
	nStatePrevious := nState;
END_IF

(*Maintance*)
IF bManualMode THEN
	nState := 150000;
END_IF

(*Emergency*)
IF NOT bEnable THEN
	nState := 0;
END_IF

(*Last states*)
IF(nState >= 1000) AND (nState < 150000) THEN
(*Steps before any state*)
	IF anLastStates[0] <> nState THEN
		FOR iLastStates:=iLastStatesMax TO 1 BY -1 DO
			anLastStates[iLastStates]:= anLastStates[iLastStates-1];
		END_FOR
		anLastStates[0]:= nState;
	END_IF
END_IF	

IF fbLift^.bError OR fbLock^.bError
THEN
	bError  :=  TRUE;
END_IF


bPalletAtStopper := fbStopper^.bPalletAtStopper;

CASE nState OF
{region "Alaphelyzet felvétel"}
	(****************************************************************************************)
	(******************************* Alaphelyzetfelvétel ************************************)
	(****************************************************************************************)	
	0:		(*-----=== Kimenetek törlése ===-----*)
		sState := CONCAT(UDINT_TO_STRING(nState) ,' - A biztonsági kör nem aktív');
		fbLift^.bBasePosCmd := FALSE;
		fbLift^.bWorkPosCmd := FALSE;
		fbLock^.bBasePosCmd := FALSE;
		fbLock^.bWorkPosCmd := FALSE;
		bError := FALSE;
		IF bEnable THEN
			IF bStepEnable THEN
				nState := nState + 20;
			END_IF
		END_IF

	20:		(*-----=== Állapotok ellenőrzése ===-----*)
		sState := CONCAT(UDINT_TO_STRING(nState) ,' - Állapotok ellenőrzése');
		IF fbLift^.i_bBasePos AND fbLock^.i_bBasePos THEN						// Lift lent és rőgzítő oldva -> Ki lehet adni az alaphelyzet vezérlést és kész
			IF bStepEnable THEN
				nState := 100;
			END_IF
		ELSE																	// Vagy fent van vagy félállapot NIMCS RÁ SZENZOR, hogy van-e nála paletta -> feltételezem, hogy van!
			IF bStepEnable THEN
				nState := 200;
			END_IF
		END_IF
	
	100:		(*-----=== Hengerek alaphelyzetbe ===-----*)
		sState := CONCAT(UDINT_TO_STRING(nState) ,' - Hengerek alaphelyzetbe');
		fbLift^.bBasePosCmd := TRUE;
		fbLift^.bWorkPosCmd := FALSE;
		fbLock^.bBasePosCmd := TRUE;
		fbLock^.bWorkPosCmd := FALSE;
		IF fbLift^.bBasePosStab AND fbLock^.bBasePosStab THEN
			IF bStepEnable THEN
				nState := 10000;
			END_IF
		END_IF

	200:		(*-----=== Hengerek munkahelyzetbe ===-----*)
		sState := CONCAT(UDINT_TO_STRING(nState) ,' - Hengerek alaphelyzetbe');
		fbLift^.bBasePosCmd := FALSE;
		fbLift^.bWorkPosCmd := TRUE;
		fbLock^.bBasePosCmd := FALSE;
		fbLock^.bWorkPosCmd := TRUE;
		IF fbLift^.bWorkPosStab AND fbLock^.bWorkPosStab THEN
			IF bStepEnable THEN
				nState := 13000;
			END_IF
		END_IF
{endregion}

{region "Alaphelyzet"}
	(****************************************************************************************)
	(*********************************** Alaphelyzet ****************************************)
	(****************************************************************************************)	
	10000:		(*-----=== Várakozás berakásra ===-----*)
		sState := CONCAT(UDINT_TO_STRING(nState) ,' - Várakozás palettára');
		IF fbStopper^.bPalletAtStopper THEN									// Paletta a stopperen
			IF bStepEnable THEN	
				nState := 11000;											// -> Alapanyag fogadása
			END_IF
		END_IF
{endregion}

{region "Alaphelyzet"}
	(****************************************************************************************)
	(*********************************** Paletta fogadása ***********************************)
	(****************************************************************************************)	
	11000:		(*-----=== RFID ellenőrzése ===-----*)
		sState := CONCAT(UDINT_TO_STRING(nState) ,' - RFID ellenőrzés');
		IF stTagData.Status <> E_TagStatus.NotPresent THEN
			IF stTagData.Code > 0 AND stTagData.Code <= 100 THEN
				IF bStepEnable THEN	
					nState := nState + 20;							// -> Valid RFID adat
				END_IF
			END_IF
		ELSIF tRFID_Timeout.Q THEN
			nState := 14000;										// -> RFID hiba -> tovább küldés
		END_IF

	11020:		(*-----=== Paletta adat ellenőrzése ===-----*)
		sState := CONCAT(UDINT_TO_STRING(nState) ,' - Paletta adat ellenőrzés');
		IF arrPaletteData^[stTagData.Code].nTarget = nReqTarget AND NOT arrPaletteData^[stTagData.Code].nState.3 THEN	
			IF bStepEnable THEN
				nTagID := stTagData.Code;						// Van darab a palettán és még nincs kész -> Kiemelés 
				nState := nState + 20;
			END_IF
		ELSE
			IF bStepEnable THEN	
				nState := 14000;								// Vagy nincs darab vagy kész -> mehet tovább
			END_IF
		END_IF

	11040:		(*-----=== Paletta rögzítése ===-----*)
		sState := CONCAT(UDINT_TO_STRING(nState) ,' - Paletta rögzítése');
		fbLock^.bBasePosCmd := FALSE;
		fbLock^.bWorkPosCmd := TRUE;
		IF fbLock^.bWorkPosStab THEN
			IF bStepEnable THEN
				nState := nState + 20;
			END_IF
		END_IF

	11060:		(*-----=== Paletta kiemelése ===-----*)
		sState := CONCAT(UDINT_TO_STRING(nState) ,' - Paletta kiemelése');
		fbLift^.bBasePosCmd := FALSE;
		fbLift^.bWorkPosCmd := TRUE;
		IF fbLift^.bWorkPosStab THEN
			IF bStepEnable THEN
				arrPaletteData^[nTagID].nState.1 := TRUE;;
				nState := 12000;
			END_IF
		END_IF
{endregion}

{region "Alaphelyzet"}
	(****************************************************************************************)
	(**************************** Várakozás megmunkálásra ***********************************)
	(****************************************************************************************)	
	12000:		(*-----=== Várakozás megmunkálásra ===-----*)
		sState := CONCAT(UDINT_TO_STRING(nState) ,' - Várakozás megmunkálásra');
		IF arrPaletteData^[nTagID].nState.3 THEN
			IF bStepEnable THEN
				arrPaletteData^[nTagID].nTarget := 0;		// Cél átírása -> Kardex
				nState := 13000;							// -> Kész a megmunkáls mehet lefelé
			END_IF
		END_IF
{endregion}

{region "Alaphelyzet"}
	(****************************************************************************************)
	(******************************** Paletta leengedése ************************************)
	(****************************************************************************************)	
	13000:		(*-----=== Paletta leengedése ===-----*)
		sState := CONCAT(UDINT_TO_STRING(nState) ,' - Paletta leengedése');
		IF NOT fbStopper^.bPalletAtStopper AND NOT bBeforeStopperSent THEN
			IF bStepEnable THEN	
				nState := nState + 20;							// Nincs a kiemelő alatt paletta -> mehet lefele
			END_IF
		END_IF

	13020:		(*-----=== Paletta leengedése ===-----*)
		sState := CONCAT(UDINT_TO_STRING(nState) ,' - Paletta leengedése');
		fbLift^.bBasePosCmd := TRUE;
		fbLift^.bWorkPosCmd := FALSE;
		IF fbLift^.bBASEPosStab THEN
			IF bStepEnable THEN
				nState := nState + 20;
			END_IF
		END_IF

	13040:		(*-----=== Paletta kioldása ===-----*)
		sState := CONCAT(UDINT_TO_STRING(nState) ,' - Paletta kioldása');
		fbLock^.bBasePosCmd := TRUE;
		fbLock^.bWorkPosCmd := FALSE;
		IF fbLock^.bBASEPosStab THEN
			IF bStepEnable THEN
				nState := nState + 20;
			END_IF
		END_IF

	13060:		(*-----=== Paletta státusz ellenőrzése ===-----*)
		sState := CONCAT(UDINT_TO_STRING(nState) ,' - Paletta státusz ellenőrzése');
		IF arrPaletteData^[nTagID].nState.3 THEN
			IF bStepEnable THEN
				nState := 14000;					// Ez egy kész darab -> Mehet a paletta elengedése
			END_IF
		ELSE
			IF bStepEnable THEN
				nState := 10000;					// Felemelt vagy félállapotú paletta(alaphelyzet felvétel)-> elleőrizni kell
			END_IF
		END_IF
{endregion}

{region "Alaphelyzet"}
	(****************************************************************************************)
	(************************ Várakozás paletta elengedésére ********************************)
	(****************************************************************************************)	
	14000:		(*-----=== Várakozás paletta elengedésére ===-----*)
		sState := CONCAT(UDINT_TO_STRING(nState) ,' - Várakozás paletta elengedésére');
		IF NOT fbStopper^.bPalletAtStopper THEN
			IF bStepEnable THEN
				nState := 10000;
			END_IF
		END_IF
{endregion}

	150000: (* Maintenance *)
		sState := CONCAT(UDINT_TO_STRING(nState) ,' - Maintenance');
		IF NOT bManualMode THEN
			nState := 0;
		END_IF
		
	200000:(* Error handling *)
		sState := CONCAT(UDINT_TO_STRING(nState) ,CONCAT(' - Error, from this state: ' , sState));
		nState := 200020;

	200020:(* Error handling *)
		IF bAckP THEN
			CASE nStatePrevious OF
				0..9999: nState := 0;
//				10000..25000: nState := 10000;
//				30000..31000: nState := 30000;
			ELSE nState := 0;
			END_CASE
		END_IF	
		
	ELSE //Not a real step, for test purposes
		sState := CONCAT(UDINT_TO_STRING(nState) ,' - Not a real step, for test purposes');
END_CASE

(*Timers***************************************************)
//fbCycleTime(IN:= nState > 10000 AND nState <= 95000, PT:= T#1D, Q=> , ET=> );
//IF nState > 10000 AND nState <= 95000 THEN
//	nCycleTime := TIME_TO_REAL(fbCycleTime.ET)/1000;
//END_IF

tRFID_Timeout(IN:= fbStopper^.bPalletAtStopper AND stTagData.Status = E_TagStatus.NotPresent, PT:= T#2s, Q=> , ET=> );

END_FUNCTION_BLOCK

// ---- POUs/FBs/Router/FB_Router.TcPOU
FUNCTION_BLOCK FB_Router
VAR_INPUT
	bEnable					: BOOL;
	bErrorAck				: BOOL;
	bManualMode				: BOOL;
	bStepEnable				: BOOL;
	stTagData				: ST_Tag_Data;
	bPaletteStopperIn		: BOOL;
	bStopperReadyBase		: BOOL;
	bStopperReadyWork		: BOOL;
	nReqTarget				: UINT;
	nNextTarget				: UINT;
END_VAR
VAR_INPUT
	fbRouter				: POINTER TO FB_Bistabil;
	arrPaletteData			: POINTER TO ARRAY [1..200] OF ST_Dut_Data;
END_VAR
VAR_OUTPUT
	nTagID					: ULINT;
END_VAR
VAR	(* Control *)
	nState						: UDINT;
	nStatePrevious				: UDINT;
	sState						: STRING(500);
	fbCycleTime					: TON;
	nCycleTime					: REAL;
	bError						: BOOL;
	tRFID_Timeout				: TON;
	tPalette					: TON;
END_VAR
VAR CONSTANT
	iLastStatesMax				: INT := 500;
END_VAR
VAR (* LastStates *)
	anLastStates				: ARRAY[0..iLastStatesMax] OF UDINT;
    iLastStates					: INT;
END_VAR

(*Error handling*)
IF nState > 0 AND nState < 150000 THEN
	nStatePrevious := nState;
END_IF

(*Maintance*)
IF bManualMode THEN
	nState := 150000;
END_IF

(*Emergency*)
IF NOT bEnable THEN
	nState := 0;
END_IF

(*Last states*)
IF(nState >= 1000) AND (nState < 150000) THEN
(*Steps before any state*)
	IF anLastStates[0] <> nState THEN
		FOR iLastStates:=iLastStatesMax TO 1 BY -1 DO
			anLastStates[iLastStates]:= anLastStates[iLastStates-1];
		END_FOR
		anLastStates[0]:= nState;
	END_IF
END_IF	

IF fbRouter^.bError
THEN
	bError  :=  TRUE;
END_IF


CASE nState OF
{region "Alaphelyzet felvétel"}
	(****************************************************************************************)
	(******************************* Alaphelyzetfelvétel ************************************)
	(****************************************************************************************)	
	0:		(*-----=== Kimenetek törlése ===-----*)
		sState := CONCAT(UDINT_TO_STRING(nState) ,' - A biztonsági kör nem aktív');
		bError := FALSE;
		IF bEnable THEN
			IF bStepEnable THEN
				nState := nState + 20;
			END_IF
			;
		END_IF

	20:		(*-----=== Állapotok ellenőrzése ===-----*)
		sState := CONCAT(UDINT_TO_STRING(nState) ,' - Állapotok ellenőrzése');
		IF fbRouter^.i_bWorkPos THEN											// Lift lent és rőgzítő oldva -> Ki lehet adni az alaphelyzet vezérlést és kész
			IF bStepEnable THEN
				nState := 200;
			END_IF
		ELSE																	// Vagy fent van vagy félállapot NIMCS RÁ SZENZOR, hogy van-e nála paletta -> feltételezem, hogy van!
			IF bStepEnable THEN
				nState := 100;
			END_IF
		END_IF
	
	100:		(*-----=== Hengerek alaphelyzetbe ===-----*)
		sState := CONCAT(UDINT_TO_STRING(nState) ,' - Hengerek alaphelyzetbe');
		fbRouter^.bBasePosCmd := TRUE;
		fbRouter^.bWorkPosCmd := FALSE;
		IF fbRouter^.bBasePosStab THEN
			IF bStepEnable THEN
				nState := 10000;				// Alaphelyzetfelvétel kész
			END_IF
		END_IF

	200:		(*-----=== Hengerek munkahelyzetbe ===-----*)
		sState := CONCAT(UDINT_TO_STRING(nState) ,' - Hengerek alaphelyzetbe');
		fbRouter^.bBasePosCmd := FALSE;
		fbRouter^.bWorkPosCmd := TRUE;
		IF fbRouter^.bWorkPosStab THEN
			IF bStepEnable THEN
				nState := 13000;				// Megkezdett folyamat befejezése
			END_IF
		END_IF
{endregion}

{region "Alaphelyzet"}
	(****************************************************************************************)
	(*********************************** Alaphelyzet ****************************************)
	(****************************************************************************************)	
	10000:		(*-----=== Várakozás palettára ===-----*)
		sState := CONCAT(UDINT_TO_STRING(nState) ,' - Várakozás palettára');
		IF bPaletteStopperIn AND stTagData.Code > 0 THEN					// Paletta a stopperen
			IF bStepEnable THEN	
				nState := 11000;											// -> Alapanyag fogadása
			END_IF
		END_IF
{endregion}

{region "Alaphelyzet"}
	(****************************************************************************************)
	(*********************************** Paletta fogadása ***********************************)
	(****************************************************************************************)	
	11000:		(*-----=== RFID ellenőrzése ===-----*)
		sState := CONCAT(UDINT_TO_STRING(nState) ,' - RFID ellenőrzés');
		IF stTagData.Status <> E_TagStatus.NotPresent THEN
			IF stTagData.Code > 0 AND stTagData.Code <= 100 THEN
				IF bStepEnable THEN
					nTagID := stTagData.Code;						// -> Valid RFID adat	
					nState := nState + 20;	
				END_IF
			END_IF
		ELSIF tRFID_Timeout.Q THEN
			nState := 13000;										// -> RFID hiba -> tovább küldés
		ELSIF NOT bPaletteStopperIn THEN
			nState := 10000;										// -> Hibás Trigger -> alaphelyzet
		END_IF

	11020:		(*-----=== Paletta adat ellenőrzése ===-----*)
		sState := CONCAT(UDINT_TO_STRING(nState) ,' - Paletta adat ellenőrzés');
		IF arrPaletteData^[nTagID].nTarget =  nReqTarget THEN	
			IF bStepEnable THEN
				nTagID := stTagData.Code;						// Target eggyezik -> leválogatás 
				nState := nState + 20;	
			END_IF
		ELSE
			IF bStepEnable THEN	
				nState := 13000;								// Vagy nincs darab vagy kész -> mehet tovább
			END_IF
		END_IF

	11040:		(*-----=== Paletta adatok frissítése ===-----*)
		sState := CONCAT(UDINT_TO_STRING(nState) ,' - Paletta adatok frissítése');
		arrPaletteData^[nTagID].nTarget := nNextTarget;
		IF bStepEnable THEN
			nState := nState + 20;
		END_IF
	
	11060:		(*-----=== Terelő munkahelyzetbe ===-----*)
		sState := CONCAT(UDINT_TO_STRING(nState) ,' - Terelő munkahelyzetbe');
		fbRouter^.bBasePosCmd := FALSE;
		fbRouter^.bWorkPosCmd := TRUE;
		IF fbRouter^.bWorkPosStab THEN
			IF bStepEnable THEN
				nState := 12000;
			END_IF
		END_IF
{endregion}

{region "Paletta elengedés"}
	(****************************************************************************************)
	(********************** Várakozás paletta elengedésre ***********************************)
	(****************************************************************************************)	
	12000:		(*-----=== Várakozás megmunkálásra ===-----*)
		sState := CONCAT(UDINT_TO_STRING(nState) ,' - Várakozás paletta elengedésre');
		IF NOT bPaletteStopperIn THEN
			IF bStepEnable THEN	
				nState := 13000;
			END_IF
		END_IF
{endregion}

{region "Paletta elhaladás"}
	(****************************************************************************************)
	(*********************** Várakozás paletta elhaladására *********************************)
	(****************************************************************************************)	
	13000:		(*-----=== Paletta elengedése ===-----*)
		sState := CONCAT(UDINT_TO_STRING(nState) ,' - Paletta elengedése');
		IF tPalette.Q THEN
			IF bStepEnable THEN	
				nState := nState + 20;
			END_IF
		END_IF

	13020:		(*-----=== Terelő alaphelyzetbe ===-----*)
		sState := CONCAT(UDINT_TO_STRING(nState) ,' - Terelő alaphelyzetbe');
		fbRouter^.bBasePosCmd := TRUE;
		fbRouter^.bWorkPosCmd := FALSE;
		IF fbRouter^.bBasePosStab THEN
			IF bStepEnable THEN
				nState := 10000;
			END_IF
		END_IF
{endregion}

	150000: (* Maintenance *)
		sState := CONCAT(UDINT_TO_STRING(nState) ,' - Maintenance');
		IF NOT bManualMode THEN
			nState := 0;
		END_IF
		
	200000:(* Error handling *)
		sState := CONCAT(UDINT_TO_STRING(nState) ,CONCAT(' - Error, from this state: ' , sState));
		nState := 200020;

	200020:(* Error handling *)
		IF bAckP THEN
			CASE nStatePrevious OF
				0..9999: nState := 0;
//				10000..25000: nState := 10000;
//				30000..31000: nState := 30000;
			ELSE nState := 0;
			END_CASE
		END_IF	
		
	ELSE //Not a real step, for test purposes
		sState := CONCAT(UDINT_TO_STRING(nState) ,' - Not a real step, for test purposes');
END_CASE

(*Timers***************************************************)
fbCycleTime(IN:= nState > 10000 AND nState <= 95000, PT:= T#1D, Q=> , ET=> );
IF nState > 10000 AND nState <= 95000 THEN
	nCycleTime := TIME_TO_REAL(fbCycleTime.ET)/1000;
END_IF

tRFID_Timeout(IN:= bPaletteStopperIn AND (stTagData.Status = E_TagStatus.NotPresent), PT:= T#2s, Q=> , ET=> );
tPalette(IN:= nState = 13000, PT:= T#2S, Q=> , ET=> );

END_FUNCTION_BLOCK

// ---- POUs/FBs/MPS/FB_MPS100.TcPOU
FUNCTION_BLOCK FB_MPS100
VAR_INPUT
	nCalOffset				: REAL;
	nReqDistance			: REAL;
	bPendantMode			: BOOL;
END_VAR
VAR_OUTPUT
	bValid					: BOOL;
	nDistance				: REAL;
	bGripperInPos			: BOOL;
END_VAR
VAR
	arrRaw		AT %I*		: ARRAY [0..1] OF BITARR8;
	nState		AT %I*		: USINT;
	nTemp					: INT;
	nAverageDistance		: REAL := 0;
	nPendantTimer			: TON;
	uConv2int				: U_to_int;
END_VAR

uConv2int.arrRaw[1] := arrRaw[0];
uConv2int.arrRaw[0] := arrRaw[1];
IF nState = 3 THEN
	bValid := TRUE;
	nTemp := SHR(uConv2int.nData,4);
	nDistance := INT_TO_REAL(nTemp)*0.05 + nCalOffset;
	nAverageDistance := (((nAverageDistance * 9) + nDistance)/10);
	IF TRUE THEN 						//bPendantMode THEN 				//megdöglött a szenzor de mennie kell midenképp!!
		bGripperInPos := nPendantTimer.Q;
	ELSE
		bGripperInPos := ABS(nDistance - nReqDistance) < 5;
	END_IF
	
ELSE
	bValid := FALSE;
	bGripperInPos := FALSE;
	nDistance := 0;
	nAverageDistance := 0;
END_IF
nPendantTimer(IN:= ABS(nAverageDistance - nDistance)< 0.5, PT:= T#500MS, Q=> , ET=> );

END_FUNCTION_BLOCK

// ---- POUs/FBs/FB_Door.TcPOU
FUNCTION_BLOCK FB_Door
VAR_INPUT
	bDoorButton			:BOOL;			// Door button imput
	bOpenEnable			:BOOL;			// The door open is possible
	bEmergencyOk		:BOOL;			// Emergency circuit state
	bWaitClose			:BOOL;			// Waiting door close 
	bDoorsClosed		:BOOL;			// Doors are closed
	bDoorsLocked		:BOOL;			// The doors are locked
	bBlink_1			:BOOL;			// Blinker for the door open button
	bBlink_2			:BOOL;			// Blinker for the cell ack button
END_VAR
VAR_OUTPUT
	bCloseOut			:BOOL;			// Door closed output
	bDoorButtonLED		:BOOL;			// Door button LED output
	bCellAckLED			:BOOL;			// Cell empty acknoledge LED output
	bObenRequestOut		:BOOL;			// Door open request output
END_VAR
VAR
	rtDoorButton		:R_Trig;		// Door open trigger
	rsOpenRequest		:RS;			// Door open request
	tOpenForce			:TON;			// Timer for forcing the doors to open
	tOpenForceDelay		:TIME := T#5S;	// Delaying for forcing the doors to open
END_VAR

(* HOW TO:
Lock: Doors are closed and the button is pushed
Open possibilities (if the doors locked and the button is pushed):
	1. Open: if the process lets the doos open
	2. Door open request register: if the process does not let the doors open, 
		from this it can go to 1, or 3rd, or it deletes the request if the button is pressed again
	3. Force open: if the button is pressed for 5 seconds, the doors open anyways *)

// Door open request
rtDoorButton(CLK:= bDoorButton);

// Lock doors
IF bEmergencyOk AND rtDoorButton.Q AND bDoorsClosed AND bWaitClose AND NOT bDoorsLocked THEN
	bCloseOut := TRUE;
END_IF

// Door open request
rsOpenRequest(
	SET:= rtDoorButton.Q AND bDoorsClosed AND bDoorsLocked, 
	RESET1:= NOT bDoorsLocked OR (rtDoorButton.Q AND rsOpenRequest.Q1),  
	Q1=> bObenRequestOut
	);

//// Door open force
//tOpenForce(IN:= bDoorButton AND bDoorsLocked, PT:= tOpenForceDelay);

// Open output
IF (rsOpenRequest.Q1 AND bOpenEnable)
	OR NOT bEmergencyOk 
//	OR tOpenForce.Q
THEN
	bCloseOut := FALSE;
END_IF

// Control for the door open blinker LED
IF bDoorsLocked THEN
	IF rsOpenRequest.Q1 THEN
		bDoorButtonLED := bBlink_1;
	ELSE
		bDoorButtonLED := TRUE;
	END_IF
ELSIF bDoorsClosed AND bWaitClose THEN
	bDoorButtonLED := bBlink_1;
ELSE
	bDoorButtonLED := FALSE;
END_IF

// Cell Ack Led
IF bEmergencyOk THEN
	IF bWaitClose THEN
		bCellAckLED := bBlink_1;
	ELSE
		bCellAckLED := bBlink_2;
	END_IF
ELSE
	bCellAckLED := FALSE;
END_IF

END_FUNCTION_BLOCK

// ---- POUs/FBs/Utilities/FB_Not_SmartLight.TcPOU
FUNCTION_BLOCK FB_Not_SmartLight
VAR_INPUT
	bEmyStop					:BOOL;
	bEmyOK						:BOOL;
	bError						:BOOL;
	bOutOfStock					:BOOL;
	bBuzzer						:BOOL;
	bBlink						:BOOL;
END_VAR
VAR_OUTPUT
	q_bGreenColor		AT %Q*	:BIT;
	q_bYellowColor		AT %Q*	:BIT;
	q_bRedColor			AT %Q*	:BIT;
	q_bBuzzer			AT %Q*	:BIT;
END_VAR
VAR
END_VAR

// Buzzzzzzzzzzzzzzzzzzzzzzzzzzzzzzzzzzzzzzzzzzzzzzzzzzzzzzz
q_bGreenColor := FALSE;
q_bYellowColor := FALSE;
q_bRedColor := FALSE;

IF bError THEN
	q_bRedColor := bBlink;
END_IF

IF bEmyOK THEN
	q_bGreenColor := TRUE;
ELSE 
	q_bGreenColor := bBlink;
END_IF

IF bOutOfStock THEN
	q_bYellowColor := bBlink;
END_IF

IF bEmyStop THEN
	q_bGreenColor := FALSE;
	q_bYellowColor := FALSE;
	q_bRedColor := TRUE;
END_IF

q_bBuzzer := bBuzzer;

END_FUNCTION_BLOCK

// ---- POUs/FBs/FB_Vise_Station.TcPOU
FUNCTION_BLOCK FB_Vise_Station
VAR_INPUT
	sName						:STRING;
	bEn							:BOOL;
	bEHA						:BOOL;
	bManualMode					:BOOL;
	bAck						:BOOL;
	sSourceName					:STRING(10);
	stViseBasePosEvent			:TcEventEntry;		(*Event definition*)
	stViseWorkPosEvent			:TcEventEntry;		(*Event definition*)
	stStopperInWorkPosEvent		:TcEventEntry;		(*Event definition*)
	stStopperOutWorkPosEvent	:TcEventEntry;		(*Event definition*)
	stViseStationSensors		:ST_Vise_Sensors;
END_VAR
VAR_OUTPUT
	bError 						:BOOL;
END_VAR
VAR
	fbVise						:FB_Bistabil;
	fbStopper_In				:FB_Bistabil;
	fbStopper_Out				:FB_Bistabil;
END_VAR

fbVise(
	sName:= sName,
	bEn:= bEn,						// AND fbStopper_In.bWorkPosStab,				Miért ?????????????????????????????????????????
	bEHA:= bEHA, 
	bDisableManualCmd:= NOT (bManualMode AND fbStopper_In.bWorkPosStab), 
	bAck:= bAckP,
	sSourceName:= sSourceName, 
	i_bBasePos:= stViseStationSensors.bViseIn,
	i_bWorkPos:= stViseStationSensors.bViseOut,
	stBasePosEvent:= stViseBasePosEvent,
	stWorkPosEvent:= stViseWorkPosEvent);
	
fbStopper_In(
	sName:= sName, 
	bEn:= bEn, 
	bEHA:= bEHA, 
	bDisableManualCmd:= NOT bManualMode, 
	bAck:= bAckP, 
	sSourceName:= sSourceName,
	i_bBasePos:= stViseStationSensors.bStopper_In_Release,
	i_bWorkPos:= stViseStationSensors.bStopper_In_Hold,
	stBasePosEvent:= TC_Events.MyEvents.Event,
	stWorkPosEvent:= stStopperInWorkPosEvent);

fbStopper_Out(
	sName:= sName, 
	bEn:= bEn, 
	bEHA:= bEHA, 
	bDisableManualCmd:= NOT bManualMode, 
	bAck:= bAckP, 
	sSourceName:= sSourceName,
	i_bBasePos:= stViseStationSensors.bStopper_Out_Release,
	i_bWorkPos:= stViseStationSensors.bStopper_Out_Hold,
	stBasePosEvent:= TC_Events.MyEvents.Event,
	stWorkPosEvent:= stStopperOutWorkPosEvent);
	
bError := fbStopper_In.bError OR fbStopper_Out.bError OR fbVise.bError;

PROPERTY PUBLIC StopperInner : REFERENCE TO FB_Bistabil
GET
StopperInner REF= fbStopper_In;
END_GET
END_PROPERTY

PROPERTY PUBLIC StopperOuter : REFERENCE TO FB_Bistabil
GET
StopperOuter REF= fbStopper_Out;
END_GET
END_PROPERTY

PROPERTY PUBLIC Vise : REFERENCE TO FB_Bistabil
GET
Vise REF= fbVise;
END_GET
END_PROPERTY

END_FUNCTION_BLOCK

// ---- POUs/FBs/Utilities/FB_RGB_Light.TcPOU
FUNCTION_BLOCK FB_RGB_Light
VAR_INPUT
	arrColors				:ARRAY [1..24] OF ST_RGB_Light;
	
END_VAR
VAR_OUTPUT
	
END_VAR
VAR
	i_stRGB_In			AT %I*	:ST_RGB_In;
	q_stRGB_Out			AT %Q*	:ST_RGB_Out;
	step						:UINT;
	i							:INT;
	n							:UINT;
	arrChannel					:ARRAY [1..24] OF UINT:=[101, 102, 103, 104, 105, 106, 107,
														201, 202, 203, 204, 205, 206, 207];
END_VAR

q_stRGB_Out.LifeSig := i_stRGB_In.LifeSig;

CASE step OF
0:
			n := 1;											// Source nr.
			q_stRGB_Out.Command := 0;
			IF i_stRGB_In.Resp = q_stRGB_Out.Command THEN
				step := step + 20;
			END_IF

20:
			FOR i:=1 TO 24 DO								// Set led colors
				IF i>=0 AND i<=6 THEN
					IF arrColors[n].nColor1State THEN
						q_stRGB_Out.arrRGB[i] := arrColors[n].nColor1;
					ELSE
						q_stRGB_Out.arrRGB[i] := 0;
					END_IF
				ELSIF i>=7 AND i<=18 THEN
					IF arrColors[n].nColor2State THEN
						q_stRGB_Out.arrRGB[i] := arrColors[n].nColor2;
					ELSE
						q_stRGB_Out.arrRGB[i] := 0;
					END_IF
				ELSIF i>=19 AND i<=24 THEN
					IF arrColors[n].nColor3State THEN
						q_stRGB_Out.arrRGB[i] := arrColors[n].nColor3;
					ELSE
						q_stRGB_Out.arrRGB[i] := 0;
					END_IF
				END_IF 
			END_FOR
			q_stRGB_Out.Command := arrChannel[n];
			step := step + 20;

40:
		IF i_stRGB_In.Resp = q_stRGB_Out.Command THEN
			n:= n + 1;
			IF n > 24 THEN
				q_stRGB_Out.Command := 10;
				step := step + 20;
			ELSE
				step := 20;
			END_IF
		END_IF

60:
		IF i_stRGB_In.Resp = q_stRGB_Out.Command THEN
			q_stRGB_Out.Command := 0;
			step := 0;
		END_IF
END_CASE

END_FUNCTION_BLOCK

// ---- POUs/FBs/Camera/FB_TCP_IP_Comm.TcPOU
FUNCTION_BLOCK FB_TCP_IP_Comm
VAR_INPUT
END_VAR
VAR_OUTPUT
END_VAR
VAR
	fbConnect 			: FB_SocketConnect;
	fbSend 				: FB_SocketSend;
	fbReceive 			: FB_SocketReceive;
	fbClose				: FB_SocketClose;
	sTxBuffer			: STRING;
	sRxBuffer			: STRING;
	sRequest			: STRING;
	sResponse			: STRING;
	sResultTmp			: STRING;
	nReadSeqStep		: INT := 0;
	nCamCheckStep		: INT := 0;

(*-----=== HMI ===-----*)
	bReadSR1000			: BOOL;
	sCode				: STRING;
	bCamCheck			: BOOL;
	rtCamReset			: R_TRIG;
	nProgNr				: UINT;
	nDimX				: LREAL;
	nDimY				: LREAL;
	nDimZ				: LREAL;
	nErrorId			: UDINT;

	_Name				:STRING;
	_RemoteHost			:STRING(15);
	_RemotePort			:UDINT;
	_ConnectTimeout		:TIME;
	_SendTimeout		:TIME;
	_ReceiveTimeout		:TIME;
	_CloseTimeout		:TIME;
	_Pass				:BOOL;
	_Fail				:BOOL;
	_Results			:ARRAY [1..10] OF STRING;
	_SavePath			:STRING(255);
	_Pos_X				:REAL;
	_Pos_Y				:REAL;
	_Pos_Z				:REAL;
	_Pos_W				:REAL;
	_Pos_P				:REAL;
	_Pos_R				:REAL;
	
END_VAR

IF bReadSR1000 THEN
	IF ReadSR1000(sCode, nErrorId) THEN
		bReadSR1000 := FALSE;
	END_IF
END_IF

rtCamReset(CLK:= bCamCheck);

IF rtCamReset.Q THEN
		ResetCam();
END_IF
IF bCamCheck THEN
	IF CamCheck(nProgNr, nDimX, nDimY, nDimZ, nErrorId) THEN
		bCamCheck := FALSE;
	END_IF
END_IF

METHOD CamCheck : BOOL
VAR_INPUT
	nProgNr		: REFERENCE TO UINT;
	nDimX		: REFERENCE TO LREAL;
	nDimY		: REFERENCE TO LREAL;
	nDimZ		: REFERENCE TO LREAL;
	nErrorId	: REFERENCE TO UDINT;
END_VAR
CamCheck := FALSE;
CASE nCamCheckStep OF
0:		_Pass := FALSE;
		_Fail := FALSE;
		sRequest := UINT_TO_STRING(nProgNr);										// Trigger parancs összeállítása
		sRequest := CONCAT('P', sRequest);
		sRequest := CONCAT(sRequest, ' [');
		sRequest := CONCAT(sRequest, LREAL_TO_STRING(nDimX));
		sRequest := CONCAT(sRequest, ';');
		sRequest := CONCAT(sRequest, LREAL_TO_STRING(nDimY));
		sRequest := CONCAT(sRequest, ';');
		sRequest := CONCAT(sRequest, LREAL_TO_STRING(nDimZ));
		sRequest := CONCAT(sRequest, ']');
		sRequest := CONCAT(sRequest, '$r$n');
		nCamCheckStep := nCamCheckStep + 20;

20:		IF ReadSequence(sRequest, sResponse, nErrorId) THEN							// Kamera kommunikáció
			_Pass := Left(sResponse,2) = Left(sRequest,2);							//Kapott válasz kiértékelése
			_Fail := NOT _Pass;
			nCamCheckStep := nCamCheckStep + 20;
		END_IF

40:		IF _Pass THEN
			sResultTmp := sResponse;												// Válasz másolása		P1 [3.206;-2.853;-130.009]$R$N  
			sResultTmp := DELETE(sResultTmp, FIND(sResultTmp, '['), 1);				// P1 [ törlése
			_Pos_X := STRING_TO_REAL(LEFT(sResultTmp, FIND(sResultTmp, ';')-1));	// X offszet másolása	3.206
			sResultTmp := DELETE(sResultTmp, FIND(sResultTmp, ';'), 1);				// X offszet törlése	3.206;
			_Pos_Y := STRING_TO_REAL(LEFT(sResultTmp, FIND(sResultTmp, ';')-1));	// Y offszet másolása	-2.853
			_Pos_Z := 0;															// Nincs használva
			_Pos_W := 0;															// Nincs használva
			_Pos_P := 0;															// Nincs használva
			sResultTmp := DELETE(sResultTmp, FIND(sResultTmp, ';'), 1);				// Y offszet törlése	-2.853;
			_Pos_R := STRING_TO_REAL(LEFT(sResultTmp, FIND(sResultTmp, ']')-1));	// Z offszet másolása	-130.009
			sResultTmp := DELETE(sResultTmp, FIND(sResultTmp, ']'), 1);				// Z offszet törlése	-130.009]
			nCamCheckStep := nCamCheckStep + 20;
		ELSE
			nCamCheckStep := nCamCheckStep + 20;
		END_IF

60:		CamCheck := TRUE;
//		nCamCheckStep := 0;															// Nincs automatikus alaphelyzet HMI miatt, trigger előtt Reset() methode hívás!
END_CASE
END_METHOD

METHOD FB_init : BOOL
VAR_INPUT
	bInitRetains : BOOL; // if TRUE, the retain variables are initialized (warm start / cold start)
	bInCopyCode : BOOL;  // if TRUE, the instance afterwards gets moved into the copy code (online change)
END_VAR
nCamCheckStep := 0;
END_METHOD

PROPERTY p_CloseTimeout :  TIME
GET
p_CloseTimeout := _CloseTimeout;
END_GET
SET
IF p_CloseTimeout > T#100MS AND p_CloseTimeout <  T#60S THEN
	_CloseTimeout := p_CloseTimeout;
ELSE
	_CloseTimeout := T#1S;					// default value
END_IF
END_SET
END_PROPERTY

PROPERTY p_ConnectTimeout : TIME
GET
p_ConnectTimeout := _ConnectTimeout;
END_GET
SET
IF p_ConnectTimeout > T#100MS AND p_ConnectTimeout <  T#60S THEN
	_ConnectTimeout := p_ConnectTimeout;
ELSE
	_ConnectTimeout := T#1S;					// default value
END_IF
END_SET
END_PROPERTY

PROPERTY p_Fail : Bool
GET
p_Fail := _Fail;
END_GET
END_PROPERTY

PROPERTY p_Name : STRING
GET
p_Name := _Name;
END_GET
SET
_Name := p_Name;
END_SET
END_PROPERTY

PROPERTY p_Pass : Bool
GET
p_Pass := _Pass;
END_GET
END_PROPERTY

PROPERTY PUBLIC p_PosP : REAL
GET
p_PosP := _Pos_P;
END_GET
END_PROPERTY

